E_SEQ_GENERAL.BUSY:;
	CASE THIS^.stSeqCtrlGeneral.iInternalSeqStateCase OF
    0:  // Nest 1 stop and low pressure pump bypass
      IF TRUE 
			AND THIS^.itfNest1.M_Stop()
      AND THIS^.itfLowPressurePump.M_Bypass(bEnable:= TRUE)
			THEN 
        PrgMeasure.bRecord := FALSE;
				THIS^.stSeqCtrlGeneral.iInternalSeqStateCase := 10; 
			END_IF
      
    10:  // Nest 2-4 stop
      IF TRUE 
			AND THIS^.itfNest2.M_Stop()
			AND THIS^.itfNest3.M_Stop()
			AND THIS^.itfNest4.M_Stop()
			THEN 
				THIS^.stSeqCtrlGeneral.iInternalSeqStateCase := 1000; 
			END_IF
      
    1000: // Exit step
      IF TRUE
      AND THIS^.itfTimerNest1.M_StopTimer()
      AND THIS^.itfTimerNest2.M_StopTimer()
      AND THIS^.itfTimerNest3.M_StopTimer()
      AND THIS^.itfTimerNest4.M_StopTimer()
			THEN 
				THIS^.stSeqCtrlGeneral.iInternalSeqStateCase := 9999; 
			END_IF
      
	ELSE
		THIS^.stSeqCtrlGeneral.eActiveSeqState := E_SEQ_GENERAL.DONE;  
	END_CASE
	THIS^.stSeqCtrlGeneral.strExtraInfo := CONCAT('Internal state: ', TO_STRING(THIS^.stSeqCtrlGeneral.iInternalSeqStateCase));
E_SEQ_GENERAL.DONE:;
E_SEQ_GENERAL.ERROR:;
E_SEQ_GENERAL.TIME_OUT:; 

IF TRUE
AND THIS^.stSeqCtrlGeneral.bTimeOutActiveQuit 
THEN
  THIS^.stSeqCtrlGeneral.strExtraInfo := 'Bitte quittieren und erneut testen';
  IF TRUE
  //AND itfOpMode.P_QUIT
  THEN
    THIS^.stSeqCtrlGeneral.eActiveSeqState := E_SEQ_GENERAL.EXECUTE;
	END_IF
  
END_IF

ELSE
  THIS^.stSeqCtrlGeneral.eActiveSeqState := E_SEQ_GENERAL.ERROR;
END_CASE
END_METHOD

METHOD PRIVATE _m_Seq_STOP_ENGINE : E_SEQ_PROCESS
VAR_INPUT
END_VAR
VAR
	ActiveSeq: STRING;
END_VAR
VAR
	
END_VAR
//THIS^._m_GeneralStepSetting(StepType:=E_STEP_STATE_TYPE.INIT,
ActiveSeq := TO_STRING(THIS^.eSeq);

CASE THIS^.stSeqCtrlGeneral.eActiveSeqState OF
E_SEQ_GENERAL.READY:;

	
E_SEQ_GENERAL.EXECUTE:;
	IF TRUE
	AND _m_Delay(T#1S)
	THEN
		THIS^.stSeqCtrlGeneral.eActiveSeqState := E_SEQ_GENERAL.RESET;
	END_IF
E_SEQ_GENERAL.RESET:;
	stSeqCtrlGeneral.iInternalSeqStateCase := 0;
  
	IF TRUE
	THEN
		THIS^.stSeqCtrlGeneral.eActiveSeqState := E_SEQ_GENERAL.BUSY;
	END_IF
E_SEQ_GENERAL.BUSY:;
	CASE THIS^.stSeqCtrlGeneral.iInternalSeqStateCase OF
		0:  // Nest 1 engine stop
      IF TRUE 
			AND THIS^.itfNest1.M_StopEngine()
			THEN 
				THIS^.stSeqCtrlGeneral.iInternalSeqStateCase := 10; 
			END_IF
      
    10: // Nest 2-4 engine stop
      IF TRUE 
			AND THIS^.itfNest2.M_StopEngine()
			AND THIS^.itfNest3.M_StopEngine()
			AND THIS^.itfNest4.M_StopEngine()
			THEN 
				THIS^.stSeqCtrlGeneral.iInternalSeqStateCase := 1000; 
			END_IF
      
    1000: // Exit step
      IF TRUE
      AND THIS^.itfTimerNest1.M_StopTimer()
      AND THIS^.itfTimerNest2.M_StopTimer()
      AND THIS^.itfTimerNest3.M_StopTimer()
      AND THIS^.itfTimerNest4.M_StopTimer()
			THEN 
				THIS^.stSeqCtrlGeneral.iInternalSeqStateCase := 9999; 
			END_IF
      
	ELSE
		THIS^.stSeqCtrlGeneral.eActiveSeqState := E_SEQ_GENERAL.DONE;  
	END_CASE
	THIS^.stSeqCtrlGeneral.strExtraInfo := CONCAT('Internal state: ', TO_STRING(THIS^.stSeqCtrlGeneral.iInternalSeqStateCase));
E_SEQ_GENERAL.DONE:;
E_SEQ_GENERAL.ERROR:;
E_SEQ_GENERAL.TIME_OUT:; 

IF TRUE
AND THIS^.stSeqCtrlGeneral.bTimeOutActiveQuit 
THEN
  THIS^.stSeqCtrlGeneral.strExtraInfo := 'Bitte quittieren und erneut testen';
  IF TRUE
  //AND itfOpMode.P_QUIT
  THEN
    THIS^.stSeqCtrlGeneral.eActiveSeqState := E_SEQ_GENERAL.EXECUTE;
	END_IF
  
END_IF

ELSE
  THIS^.stSeqCtrlGeneral.eActiveSeqState := E_SEQ_GENERAL.ERROR;
END_CASE
END_METHOD

METHOD PRIVATE _m_SequenceManager
VAR_INPUT
END_VAR
IF FALSE
//AND THIS^.eActiveSeqState=DONE 
AND eLastSeq<>eSeq
THEN
	IF THIS^.stSeqCtrlGeneral.eActiveSeqState<>E_SEQ_GENERAL.EXECUTE THEN
		THIS^.stSeqCtrlGeneral.eActiveSeqState:=E_SEQ_GENERAL.READY;
	END_IF
END_IF

eSeq := eNextSeq;

//DelayTimer und TimeOut Timer verwalten
stSeqCtrlGeneral.bActiveStep:=	TRUE
				AND eLastSeq					=	eSeq
				AND stSeqCtrlGeneral.eLastActiveSeqState			=	stSeqCtrlGeneral.eActiveSeqState
				AND	stSeqCtrlGeneral.iLastInternalSeqStateCase	=	stSeqCtrlGeneral.iInternalSeqStateCase
				;
			
IF NOT stSeqCtrlGeneral.bActiveStep THEN
	stSeqCtrlGeneral.bDelayActive:=FALSE;
	stSeqCtrlGeneral.bTimeOutActiveQuit:=FALSE;
	stSeqCtrlGeneral.bTimeOutActiveNoQuit:=FALSE;
  THIS^.stSeqCtrlGeneral.strExtraInfo:='';
END_IF

_m_SaveLastStep();
stSeqCtrlGeneral.tonDelay	(IN:=stSeqCtrlGeneral.bActiveStep AND stSeqCtrlGeneral.bDelayActive, 		PT:=stSeqCtrlGeneral.tDelay);
stSeqCtrlGeneral.tonTimeOut	(IN:=stSeqCtrlGeneral.bActiveStep AND (stSeqCtrlGeneral.bTimeOutActiveNoQuit OR stSeqCtrlGeneral.bTimeOutActiveQuit), 	PT:=stSeqCtrlGeneral.tTimeOut);
stSeqCtrlGeneral.tonStepTime	(IN:= stSeqCtrlGeneral.bActiveStep, PT:= T#24H);

IF stSeqCtrlGeneral.tonTimeOut.Q  THEN
	stSeqCtrlGeneral.eActiveSeqState:=E_SEQ_GENERAL.TIME_OUT;
END_IF

IF stSeqCtrlGeneral.iError<>0 THEN
	eSeq:=E_SEQ_PROCESS.ERROR_SEQ;
END_IF



eLastSeq					:=	eSeq;
stSeqCtrlGeneral.eLastActiveSeqState			:=	stSeqCtrlGeneral.eActiveSeqState;
stSeqCtrlGeneral.iLastInternalSeqStateCase	:=	stSeqCtrlGeneral.iInternalSeqStateCase;

// Reset set ready state
IF THIS^.stSeqCtrlGeneral.bExitSetReadyState THEN
  THIS^.stSeqCtrlGeneral.bExitSetReadyState := FALSE;
END_IF
END_METHOD

METHOD PRIVATE _m_TimeOut : BOOL
VAR_INPUT
	bTimeoutActiveToQuit:	BOOL;
	bTimeOutActiveNoQuit:	BOOL;
	tTimeOut:				TIME;	
END_VAR
THIS^.stSeqCtrlGeneral.bTimeOutActiveQuit:=	bTimeoutActiveToQuit;
THIS^.stSeqCtrlGeneral.bTimeOutActiveNoQuit:=	bTimeOutActiveNoQuit;
THIS^.stSeqCtrlGeneral.tTimeOut:=			tTimeOut;
_m_TimeOut:=FALSE;
IF THIS^.stSeqCtrlGeneral.tonTimeOut.Q THEN
	_m_TimeOut:=TRUE;
END_IF
END_METHOD

METHOD FB_init : BOOL
VAR_INPUT
	bInitRetains : BOOL; // if TRUE, the retain variables are initialized (warm start / cold start)
	bInCopyCode : BOOL;  // if TRUE, the instance afterwards gets moved into the copy code (online change)
  
  itfOpMode:											                        I_OP_MODE; 
  itfEventLogger:                                         I_EVENT_LOGGER; 
  itfTimerNest1:                                          I_CLOCK; 
  itfTimerNest2:                                          I_CLOCK; 
  itfTimerNest3:                                          I_CLOCK; 
  itfTimerNest4:                                          I_CLOCK;
  itfNest1:                                               I_PROCESS_NEST1;
  itfNest2:                                               I_PROCESS_NEST2_4;
  itfNest3:                                               I_PROCESS_NEST2_4;
  itfNest4:                                               I_PROCESS_NEST2_4;
  itfLowPressurePump:                                     I_PUMP_WITH_BYPASS;
  itfOilCooler:                                           I_PUMP;
  itfBypassPump:                                          I_PUMP;
  itfLevelSwitch_AggregateTank1_Out1:                     I_BINARY_SWITCH;
  itfLevelSwitch_AggregateTank1_Out2:                     I_BINARY_SWITCH;
  itfTemperatureSwitch_AggregateTank1_Out1:               I_BINARY_SWITCH;
  itfTemperatureSwitch_AggregateTank1_Out2:               I_BINARY_SWITCH;
  itfLevelSwitch_AggregateTank2_Out1:                     I_BINARY_SWITCH;
  itfLevelSwitch_AggregateTank2_Out2:                     I_BINARY_SWITCH;
  itfLevelSwitch_AggregateTank2_Out3:                     I_BINARY_SWITCH;
  itfSwitch_AggregateFilter_Dirty:                        I_BINARY_SWITCH; 
END_VAR
THIS^.itfOpMode := itfOpMode;
THIS^.itfEventLogger := itfEventLogger;
THIS^.itfTimerNest1 := itfTimerNest1;
THIS^.itfTimerNest2 := itfTimerNest2;
THIS^.itfTimerNest3 := itfTimerNest3;
THIS^.itfTimerNest4 := itfTimerNest4;
THIS^.itfNest1 := itfNest1;
THIS^.itfNest2 := itfNest2;
THIS^.itfNest3 := itfNest3;
THIS^.itfNest4 := itfNest4;
THIS^.itfLowPressurePump := itfLowPressurePump;
THIS^.itfOilCooler := itfOilCooler;
THIS^.itfBypassPump := itfBypassPump;
THIS^.itfLevelSwitch_AggregateTank1_Out1 := itfLevelSwitch_AggregateTank1_Out1;
THIS^.itfLevelSwitch_AggregateTank1_Out2 := itfLevelSwitch_AggregateTank1_Out2;
THIS^.itfTemperatureSwitch_AggregateTank1_Out1 := itfTemperatureSwitch_AggregateTank1_Out1;
THIS^.itfTemperatureSwitch_AggregateTank1_Out2 := itfTemperatureSwitch_AggregateTank1_Out2;
THIS^.itfLevelSwitch_AggregateTank2_Out1 := itfLevelSwitch_AggregateTank2_Out1;
THIS^.itfLevelSwitch_AggregateTank2_Out2 := itfLevelSwitch_AggregateTank2_Out2;
THIS^.itfLevelSwitch_AggregateTank2_Out3 := itfLevelSwitch_AggregateTank2_Out3;
THIS^.itfSwitch_AggregateFilter_Dirty := itfSwitch_AggregateFilter_Dirty;
END_METHOD

METHOD M_BreakPressureDet : BOOL
VAR_INPUT
  stBreakPressureParams:                 ST_RECIPE_BREAK_PRESSURE;
END_VAR
M_BreakPressureDet := THIS^.stSeqCtrlGeneral.eActiveSeqState = E_SEQ_GENERAL.DONE;

// Assign input
THIS^.stBPDParams := stBreakPressureParams;

// General
IF THIS^.stSeqCtrlGeneral.eActiveSeqState = E_SEQ_GENERAL.READY THEN
  THIS^.eNextSeq := E_SEQ_PROCESS.BREAK_PRESSURE_DET;
  THIS^.stSeqCtrlGeneral.eActiveSeqState := E_SEQ_GENERAL.EXECUTE;
END_IF
END_METHOD

METHOD M_EnduranceRun : BOOL
VAR_INPUT
  stEnduranceRunParams:                 ST_RECIPE_ENDURANCE_RUN;
END_VAR
M_EnduranceRun := THIS^.stSeqCtrlGeneral.eActiveSeqState = E_SEQ_GENERAL.DONE;

// Assign input
THIS^.stERParams := stEnduranceRunParams;

// General
IF THIS^.stSeqCtrlGeneral.eActiveSeqState = E_SEQ_GENERAL.READY THEN
  THIS^.eNextSeq := E_SEQ_PROCESS.ENDURANCE_RUN;
  THIS^.stSeqCtrlGeneral.eActiveSeqState := E_SEQ_GENERAL.EXECUTE;
END_IF
END_METHOD

METHOD M_EStop : BOOL
M_EStop := THIS^.stSeqCtrlGeneral.eActiveSeqState = E_SEQ_GENERAL.DONE;

IF THIS^.stSeqCtrlGeneral.eActiveSeqState = E_SEQ_GENERAL.READY THEN
  THIS^.eNextSeq := E_SEQ_PROCESS.ESTOP;
  THIS^.stSeqCtrlGeneral.eActiveSeqState := E_SEQ_GENERAL.EXECUTE;
END_IF
END_METHOD

METHOD M_LeakTest1 : BOOL
VAR_INPUT
  stLeakTest1Params:                 ST_RECIPE_LEAK_TEST1;
END_VAR
M_LeakTest1 := THIS^.stSeqCtrlGeneral.eActiveSeqState = E_SEQ_GENERAL.DONE;

// Assign input
THIS^.stLT1Params := stLeakTest1Params;

// General
IF THIS^.stSeqCtrlGeneral.eActiveSeqState = E_SEQ_GENERAL.READY THEN
  THIS^.eNextSeq := E_SEQ_PROCESS.LEAK_TEST_1;
  THIS^.stSeqCtrlGeneral.eActiveSeqState := E_SEQ_GENERAL.EXECUTE;
END_IF
END_METHOD

METHOD M_LeakTest2 : BOOL
VAR_INPUT
  stLeakTest2Params:                 ST_RECIPE_LEAK_TEST2;
END_VAR
M_LeakTest2 := THIS^.stSeqCtrlGeneral.eActiveSeqState = E_SEQ_GENERAL.DONE;

// Assign input
THIS^.stLT2Params := stLeakTest2Params;

// General
IF THIS^.stSeqCtrlGeneral.eActiveSeqState = E_SEQ_GENERAL.READY THEN
  THIS^.eNextSeq := E_SEQ_PROCESS.LEAK_TEST_2;
  THIS^.stSeqCtrlGeneral.eActiveSeqState := E_SEQ_GENERAL.EXECUTE;
END_IF
END_METHOD

METHOD M_Reset : BOOL
M_Reset := THIS^.stSeqCtrlGeneral.eActiveSeqState = E_SEQ_GENERAL.DONE;

IF THIS^.stSeqCtrlGeneral.eActiveSeqState = E_SEQ_GENERAL.READY THEN
  THIS^.eNextSeq := E_SEQ_PROCESS.INIT;
  THIS^.stSeqCtrlGeneral.eActiveSeqState := E_SEQ_GENERAL.EXECUTE;
END_IF
END_METHOD

{warning 'Methodenimplementierung hinzufügen'}
(*=== Method: M_Run  ============================================

 @brief: Here is the global code (Timer, Event, Flange,...)*)
METHOD M_Run
END_METHOD

METHOD M_SetReady : BOOL
VAR_INPUT
  
END_VAR
M_SetReady := TRUE
              AND THIS^.stSeqCtrlGeneral.eActiveSeqState = E_SEQ_GENERAL.READY
              AND THIS^.eSeq = E_SEQ_PROCESS.BASE;

THIS^.stSeqCtrlGeneral.eActiveSeqState := E_SEQ_GENERAL.READY;
THIS^.eNextSeq := E_SEQ_PROCESS.BASE;
END_METHOD

METHOD M_Stop : BOOL
M_Stop := THIS^.stSeqCtrlGeneral.eActiveSeqState = E_SEQ_GENERAL.DONE;

IF THIS^.stSeqCtrlGeneral.eActiveSeqState = E_SEQ_GENERAL.READY THEN
  THIS^.eNextSeq := E_SEQ_PROCESS.STOP;
  THIS^.stSeqCtrlGeneral.eActiveSeqState := E_SEQ_GENERAL.EXECUTE;
END_IF
END_METHOD

METHOD M_StopEngine : BOOL
M_StopEngine := THIS^.stSeqCtrlGeneral.eActiveSeqState = E_SEQ_GENERAL.DONE;

IF THIS^.stSeqCtrlGeneral.eActiveSeqState = E_SEQ_GENERAL.READY THEN
  THIS^.eNextSeq := E_SEQ_PROCESS.STOP_ENGINE;
  THIS^.stSeqCtrlGeneral.eActiveSeqState := E_SEQ_GENERAL.EXECUTE;
END_IF
END_METHOD

{warning 'Eigenschaftenimplementierung hinzufügen'}
PROPERTY P_CurrentCycleNest1 : UDINT
GET
P_CurrentCycleNest1 := THIS^.udiCurrentCyclesNest1;
END_GET
END_PROPERTY

{warning 'Eigenschaftenimplementierung hinzufügen'}
PROPERTY P_CurrentCycleNest2 : UDINT
GET
P_CurrentCycleNest2 := THIS^.udiCurrentCyclesNest2;
END_GET
END_PROPERTY

{warning 'Eigenschaftenimplementierung hinzufügen'}
PROPERTY P_CurrentCycleNest3 : UDINT
GET
P_CurrentCycleNest3 := THIS^.udiCurrentCyclesNest3;
END_GET
END_PROPERTY

{warning 'Eigenschaftenimplementierung hinzufügen'}
PROPERTY P_CurrentCycleNest4 : UDINT
GET
P_CurrentCycleNest4 := THIS^.udiCurrentCyclesNest4;
END_GET
END_PROPERTY

{warning 'Eigenschaftenimplementierung hinzufügen'}
(*=== Property: P_Event  ============================================

 @param [set]: 	Set the Structure "ST_EVENT" from another Object
 @param [get]: 	Return the Structure "ST_EVENT", it contains the actual 
					event of the Object *)
PROPERTY P_Event : GenLib.ST_EVENT
GET
END_GET
SET
END_SET
END_PROPERTY

{warning 'Eigenschaftenimplementierung hinzufügen'}
(*=== Property: P_FullObjectPath  ============================================

 @param [set]: 	Set the Object Path (Clear String of Object)
 @param [get]: 	Return the Objectpath *)
PROPERTY P_FullObjectPath : STRING
GET
END_GET
SET
END_SET
END_PROPERTY

{warning 'Eigenschaftenimplementierung hinzufügen'}
(*=== Property: P_Global_Ack  ============================================

 @param [set]: 	Set the Bit for Ack from another Object
 @param [get]: 	Return the state of Ack Bit*)
PROPERTY P_Global_Ack : BOOL
GET
END_GET
SET
END_SET
END_PROPERTY

{warning 'Eigenschaftenimplementierung hinzufügen'}
(*=== Property: P_GlobalID  ============================================

 @param [set]: 	-
 @param [get]: 	Return the string of instance path*)
PROPERTY P_GlobalID : STRING
GET
END_GET
END_PROPERTY

{warning 'Eigenschaftenimplementierung hinzufügen'}
PROPERTY P_ReadyState : BOOL
GET
P_ReadyState := THIS^.stSeqCtrlGeneral.eActiveSeqState = E_SEQ_GENERAL.READY;
END_GET
END_PROPERTY

END_FUNCTION_BLOCK

// ---- FUNCTIONS/FUNCTIONS/MATH/F_RoundLREAL.TcPOU
FUNCTION F_RoundLREAL : LREAL
VAR_INPUT
	lrValue:					LREAL;
	uiDezimalPlace:	UINT;
END_VAR
VAR
	lrResult:				REAL;
	uiMultiplier:		UINT := 1;
	i:							UINT;
END_VAR

FOR i := 1 TO uiDezimalPlace BY 1 DO
	uiMultiplier := uiMultiplier * 10;
END_FOR

lrResult := TO_REAL(TO_DINT(lrValue * uiMultiplier)) / uiMultiplier;

F_RoundLREAL := lrResult;

END_FUNCTION

// ---- MODULE/ACTOR_VALVE/PNEUMATIC_ACTOR/POU/FB_STOP_GATE.TcPOU
{attribute 'reflection'} 
{attribute 'no_explicit_call' := 'do not call this POU directly'} 
FUNCTION_BLOCK FB_STOP_GATE IMPLEMENTS I_STOP_GATE
VAR_INPUT
END_VAR
VAR_OUTPUT
END_VAR
VAR
	{attribute 'instance-path'} 
    {attribute 'noinit'} 
	strInstancePath: STRING;
	strFullObjectPath: STRING;
	stEvent: ST_EVENT;
	bAck: BOOL;
	itfOpMode:				I_OP_MODE;
	itfValveOpenStopGate:	I_BASE_VALVE;
	itfSensorByStopGate: 	I_BINARY_SWITCH;
	itfSensorCongestion: 	I_BINARY_SWITCH;
	
	tonToBase: Tc2_Standard.TON;
	tToBase: TIME;
	tonToWork: Tc2_Standard.TON;
	tToWork: TIME;
	bViewToBase: BOOL;
	bViewToWork: BOOL;
	
	
END_VAR

METHOD FB_init : BOOL
VAR_INPUT
	bInitRetains : BOOL; // if TRUE, the retain variables are initialized (warm start / cold start)
	bInCopyCode : BOOL;  // if TRUE, the instance afterwards gets moved into the copy code (online change)
END_VAR
END_METHOD

{warning 'Methodenimplementierung hinzufügen'}
METHOD M_Close
END_METHOD

{warning 'Methodenimplementierung hinzufügen'}
METHOD M_Open
END_METHOD

{warning 'Methodenimplementierung hinzufügen'}
(*=== Method: M_Run  ============================================

 @brief: Here is the global code (Timer, Event, Flange,...)*)
METHOD M_Run
END_METHOD

{warning 'Methodenimplementierung hinzufügen'}
METHOD M_Seperate
VAR_INPUT
	iCntCarrier	: INT;
END_VAR
END_METHOD


PROPERTY P_CarrierByStopGate : BOOL
GET
END_GET
END_PROPERTY


PROPERTY P_Congestion : BOOL
GET
END_GET
END_PROPERTY


(*=== Property: P_Event  ============================================

 @param [set]: 	Set the Structure "ST_EVENT" from another Object
 @param [get]: 	Return the Structure "ST_EVENT", it contains the actual 
					event of the Object *)
PROPERTY P_Event : ST_EVENT
GET
END_GET
SET
END_SET
END_PROPERTY


(*=== Property: P_FullObjectPath  ============================================

 @param [set]: 	Set the Object Path (Clear String of Object)
 @param [get]: 	Return the Objectpath *)
PROPERTY P_FullObjectPath : STRING
GET
END_GET
SET
END_SET
END_PROPERTY


(*=== Property: P_Global_Ack  ============================================

 @param [set]: 	Set the Bit for Ack from another Object
 @param [get]: 	Return the state of Ack Bit*)
PROPERTY P_Global_Ack : BOOL
GET
END_GET
SET
END_SET
END_PROPERTY


(*=== Property: P_GlobalID  ============================================

 @param [set]: 	-
 @param [get]: 	Return the string of instance path*)
PROPERTY P_GlobalID : STRING
GET
END_GET
END_PROPERTY

END_FUNCTION_BLOCK

// ---- MODULE/ACTOR_VALVE/PNEUMATIC_ACTOR/POU/FB_VAC_BLOW_VALVE.TcPOU
{attribute 'reflection'} 
{attribute 'no_explicit_call' := 'do not call this POU directly'} 
FUNCTION_BLOCK FB_VAC_BLOW_VALVE IMPLEMENTS I_VAC_VALVE
VAR_INPUT
END_VAR
VAR_OUTPUT
END_VAR
VAR
	{attribute 'instance-path'} 
    {attribute 'noinit'} 
	strInstancePath: STRING;
	strFullObjectPath: STRING;
	stEvent: ST_EVENT;
	bAck: BOOL;
	itfOpMode:			I_OP_MODE;
	itfValveVac: I_BASE_VALVE;
	itfValveBlow: I_BASE_VALVE;
	itfSensorVacDetect: I_BINARY_SWITCH;

	
END_VAR

METHOD FB_init : BOOL
VAR_INPUT
	bInitRetains : BOOL; // if TRUE, the retain variables are initialized (warm start / cold start)
	bInCopyCode : BOOL;  // if TRUE, the instance afterwards gets moved into the copy code (online change)
	itfOpMode:			I_OP_MODE;
	itfValveVac: I_BASE_VALVE;
	itfValveBlow: I_BASE_VALVE;
	itfSensorVacDetect: I_BINARY_SWITCH;
END_VAR
THIS^.itfOpMode:= itfOpMode;
THIS^.itfValveVac:= itfValveVac;
THIS^.itfValveBlow:= itfValveBlow;
THIS^.itfSensorVacDetect:= itfSensorVacDetect;
END_METHOD

{warning 'Methodenimplementierung hinzufügen'}
METHOD M_AllOff
THIS^.itfValveVac.M_Close();
THIS^.itfValveBlow.M_Close();
END_METHOD

{warning 'Methodenimplementierung hinzufügen'}
METHOD M_Blow
THIS^.itfValveVac.M_Close();
THIS^.itfValveBlow.M_OPEN();
END_METHOD

{warning 'Methodenimplementierung hinzufügen'}
(*=== Method: M_Run  ============================================

 @brief: Here is the global code (Timer, Event, Flange,...)*)
METHOD M_Run
F_HandleInheritanceObjectInMRun(itfInheritanceObject:=THIS^.itfSensorVacDetect,itfThisObject:=THIS^);
F_HandleInheritanceObjectInMRun(itfInheritanceObject:=THIS^.itfValveVac,itfThisObject:=THIS^);
END_METHOD

{warning 'Methodenimplementierung hinzufügen'}
METHOD M_Vac
THIS^.itfValveVac.M_OPEN();
THIS^.itfValveBlow.M_Close();
END_METHOD


(*=== Property: P_Event  ============================================

 @param [set]: 	Set the Structure "ST_EVENT" from another Object
 @param [get]: 	Return the Structure "ST_EVENT", it contains the actual 
					event of the Object *)
PROPERTY P_Event : ST_EVENT
GET
P_Event:= stEvent;
END_GET
SET
END_SET
END_PROPERTY


(*=== Property: P_FullObjectPath  ============================================

 @param [set]: 	Set the Object Path (Clear String of Object)
 @param [get]: 	Return the Objectpath *)
PROPERTY P_FullObjectPath : STRING
GET
P_FullObjectPath:= THIS^.strFullObjectPath;
END_GET
SET
THIS^.strFullObjectPath:= P_FullObjectPath;
END_SET
END_PROPERTY


(*=== Property: P_Global_Ack  ============================================

 @param [set]: 	Set the Bit for Ack from another Object
 @param [get]: 	Return the state of Ack Bit*)
PROPERTY P_Global_Ack : BOOL
GET
P_Global_Ack:= THIS^.bAck;
END_GET
SET
THIS^.bAck:=P_Global_Ack;
END_SET
END_PROPERTY


(*=== Property: P_GlobalID  ============================================

 @param [set]: 	-
 @param [get]: 	Return the string of instance path*)
PROPERTY P_GlobalID : STRING
GET
P_GlobalID:= THIS^.strInstancePath;
END_GET
END_PROPERTY


PROPERTY P_STATE : E_PNEU_VAC_VALVE
GET
IF THIS^.itfValveVac.P_IS_OPEN THEN
	P_STATE:=E_PNEU_VAC_VALVE.Vac_ON_NotDetect;
END_IF

IF THIS^.itfValveVac.P_IS_CLOSE THEN
	P_STATE:=E_PNEU_VAC_VALVE.AllOff;
END_IF

IF THIS^.itfSensorVacDetect.P_Active THEN
	 P_STATE:=E_PNEU_VAC_VALVE.VacDetect;
 END_IF
 
 IF THIS^.itfValveBlow.P_IS_OPEN THEN
	 P_STATE:=E_PNEU_VAC_VALVE.Blowing;
 END_IF
END_GET
END_PROPERTY

END_FUNCTION_BLOCK

// ---- MODULE/ACTOR_VALVE/PNEUMATIC_ACTOR/POU/FB_VAC_VALVE.TcPOU
{attribute 'reflection'} 
{attribute 'no_explicit_call' := 'do not call this POU directly'} 
FUNCTION_BLOCK FB_VAC_VALVE IMPLEMENTS I_VAC_VALVE
VAR_INPUT
END_VAR
VAR_OUTPUT
END_VAR
VAR
	{attribute 'instance-path'} 
    {attribute 'noinit'} 
	strInstancePath: STRING;
	strFullObjectPath: STRING;
	stEvent: ST_EVENT;
	bAck: BOOL;
	itfOpMode:			I_OP_MODE;
	itfValveVac: I_BASE_VALVE;
	itfSensorVacDetect: I_BINARY_SWITCH;

	
END_VAR

METHOD FB_init : BOOL
VAR_INPUT
	bInitRetains : BOOL; // if TRUE, the retain variables are initialized (warm start / cold start)
	bInCopyCode : BOOL;  // if TRUE, the instance afterwards gets moved into the copy code (online change)
	itfOpMode:	I_OP_MODE;
	itfValveVac: I_BASE_VALVE;
	itfSensorVacDetect: I_BINARY_SWITCH;
END_VAR
THIS^.itfOpMode:= itfOpMode;
THIS^.itfValveVac:= itfValveVac;
THIS^.itfSensorVacDetect:= itfSensorVacDetect;
END_METHOD

{warning 'Methodenimplementierung hinzufügen'}
METHOD M_AllOff
THIS^.itfValveVac.M_Close();
END_METHOD

{warning 'Methodenimplementierung hinzufügen'}
METHOD M_Blow
THIS^.itfValveVac.M_Close();
END_METHOD

{warning 'Methodenimplementierung hinzufügen'}
(*=== Method: M_Run  ============================================

 @brief: Here is the global code (Timer, Event, Flange,...)*)
METHOD M_Run
F_HandleInheritanceObjectInMRun(itfInheritanceObject:=THIS^.itfSensorVacDetect,itfThisObject:=THIS^);
F_HandleInheritanceObjectInMRun(itfInheritanceObject:=THIS^.itfValveVac,itfThisObject:=THIS^);
END_METHOD

{warning 'Methodenimplementierung hinzufügen'}
METHOD M_Vac
THIS^.itfValveVac.M_OPEN();
END_METHOD


(*=== Property: P_Event  ============================================

 @param [set]: 	Set the Structure "ST_EVENT" from another Object
 @param [get]: 	Return the Structure "ST_EVENT", it contains the actual 
					event of the Object *)
PROPERTY P_Event : ST_EVENT
GET
P_Event:= stEvent;
END_GET
SET
END_SET
END_PROPERTY


(*=== Property: P_FullObjectPath  ============================================

 @param [set]: 	Set the Object Path (Clear String of Object)
 @param [get]: 	Return the Objectpath *)
PROPERTY P_FullObjectPath : STRING
GET
P_FullObjectPath:= THIS^.strFullObjectPath;
END_GET
SET
THIS^.strFullObjectPath:= P_FullObjectPath;
END_SET
END_PROPERTY


(*=== Property: P_Global_Ack  ============================================

 @param [set]: 	Set the Bit for Ack from another Object
 @param [get]: 	Return the state of Ack Bit*)
PROPERTY P_Global_Ack : BOOL
GET
P_Global_Ack:= THIS^.bAck;
END_GET
SET
THIS^.bAck:=P_Global_Ack;
END_SET
END_PROPERTY


(*=== Property: P_GlobalID  ============================================

 @param [set]: 	-
 @param [get]: 	Return the string of instance path*)
PROPERTY P_GlobalID : STRING
GET
P_GlobalID:= THIS^.strInstancePath;
END_GET
END_PROPERTY


PROPERTY P_STATE : E_PNEU_VAC_VALVE
GET
IF THIS^.itfValveVac.P_IS_OPEN THEN
	P_STATE:=E_PNEU_VAC_VALVE.Vac_ON_NotDetect;
END_IF

IF THIS^.itfValveVac.P_IS_CLOSE THEN
	P_STATE:=E_PNEU_VAC_VALVE.AllOff;
END_IF

IF THIS^.itfSensorVacDetect.P_Active THEN
	 P_STATE:=E_PNEU_VAC_VALVE.VacDetect;
 END_IF
END_GET
END_PROPERTY

END_FUNCTION_BLOCK

// ---- MODULE/ACTOR_VALVE/PNEUMATIC_ACTOR/POU/FB_VISU_CYLINDER.TcPOU
FUNCTION_BLOCK FB_VISU_CYLINDER
VAR_INPUT
END_VAR
VAR_OUTPUT
END_VAR
VAR
	itfPneuActor: I_PNEU_ACTOR;	
	itfOpMode: I_OP_MODE;
	iMove: INT;
	iNegMove: INT;
	iMoveSmall: INT;
	iNegMoveSmall: INT;
	iAngle: INT;
	iNegAngle: INT;
	strInfo: STRING;
	strFullObjName: STRING;
	bMoveToBase: BOOL;
	bMoveToWork: BOOL;
	bAllOff: BOOL;
	bInBasePos: BOOL;
	bInWorkPos: BOOL;
	bInMidPos: 	BOOL;
	bFaultWorkPos: BOOL;
	bFaultBasePos: BOOL;
	dwFrameColorBase: DWORD:= 16#FF00BFFF;
	dwFrameColorWork: DWORD:= 16#FF00BFFF;
	dwFrameColorMid: DWORD:= 16#FF00BFFF;
	bBaseArrowInvisible: BOOL:=TRUE;
	bWorkArrowInvisible: BOOL:=TRUE;
	bMidkArrowInvisible: BOOL:=TRUE;
	iFrame: INT;
	bFrameInvisible: BOOL:= TRUE;
	stEvent: ST_EVENT;
	dwColor: DWORD;
END_VAR

IF NOT (itfOpMode.P_OP_MODE_STATE=OP_MODE.MANUAL) THEN
	bFrameInvisible:= TRUE;
END_IF

IF (itfPneuActor.P_State=E_POS_STATE.MoveToBase) THEN
//IF bMoveToBase AND NOT bInBasePos THEN
	iMove:=-30;
	iAngle:=-90;
	//strInfo:= 'Zylinder fährt in Grundposition';
	strInfo:= F_RET_TXTLIST_ENTRY(strPortNr:= '851', strID:='3', strTxtLstName:= 'TXT_LIST_PNEMATIC_ACTOR');
	//bMoveToWork:= FALSE;
	dwFrameColorBase:= 16#FFFFA500;
	bBaseArrowInvisible:= FALSE;
	bWorkArrowInvisible:=TRUE;	
	bMidkArrowInvisible:=TRUE;
END_IF

IF (itfPneuActor.P_State=E_POS_STATE.InBasePos) THEN
//IF bMoveToBase AND bInBasePos THEN
	iMove:=0;
	iAngle:=0;
	//strInfo:= 'Zylinder ist in Grundposition';
	strInfo:= F_RET_TXTLIST_ENTRY(strPortNr:= '851', strID:='4', strTxtLstName:= 'TXT_LIST_PNEMATIC_ACTOR');
	//bMoveToWork:= FALSE;
	dwFrameColorBase:= 16#FF77BB77;
	bBaseArrowInvisible:= FALSE;
	bWorkArrowInvisible:=TRUE;	
	bMidkArrowInvisible:=TRUE;
END_IF

IF (itfPneuActor.P_State=E_POS_STATE.MoveToWork) THEN
//IF bMoveToWork AND NOT bInworkPos THEN
	iMove:=-30;
	iAngle:=-90;
	//strInfo:= 'Zylinder fährt in Arbeitsposition';
	strInfo:= F_RET_TXTLIST_ENTRY(strPortNr:= '851', strID:='5', strTxtLstName:= 'TXT_LIST_PNEMATIC_ACTOR');
	//bMoveToBase:= FALSE;
	dwFrameColorwork:= 16#FFFFA500;
	bBaseArrowInvisible:= TRUE;
	bWorkArrowInvisible:=FALSE;	
	bMidkArrowInvisible:=TRUE;
END_IF

IF (itfPneuActor.P_State=E_POS_STATE.InWorkPos) THEN
//IF bMoveToWork AND bInWorkPos THEN
	iMove:=-70;
	iAngle:=180;
	//strInfo:= 'Zylinder ist in Arbeitsposition';
	strInfo:= F_RET_TXTLIST_ENTRY(strPortNr:= '851', strID:='6', strTxtLstName:= 'TXT_LIST_PNEMATIC_ACTOR');
	//bMoveTobase:= FALSE;
	dwFrameColorWork:= 16#FF77BB77;
	bBaseArrowInvisible:= TRUE;
	bWorkArrowInvisible:=FALSE;	
	bMidkArrowInvisible:=TRUE;
END_IF

IF (itfPneuActor.P_State=E_POS_STATE.InMidPos) THEN
//IF bMoveToWork AND bInWorkPos THEN
	iMove:=-50;
	iAngle:=-90;
	//strInfo:= 'Zylinder ist in Arbeitsposition';
	strInfo:= F_RET_TXTLIST_ENTRY(strPortNr:= '851', strID:='15', strTxtLstName:= 'TXT_LIST_PNEMATIC_ACTOR');
	//bMoveTobase:= FALSE;
	dwFrameColorMid:= 16#FF77BB77;
	bBaseArrowInvisible:= TRUE;
	bWorkArrowInvisible:=TRUE;	
	bMidkArrowInvisible:=FALSE;
END_IF

IF (itfPneuActor.P_State=E_POS_STATE.NoDefPos) THEN
//IF bMoveToWork AND bInWorkPos THEN
	iMove:=-30;
	iNegAngle:=-90;
	//strInfo:= 'Zylinder in undefinierter Position';
	strInfo:= F_RET_TXTLIST_ENTRY(strPortNr:= '851', strID:='7', strTxtLstName:= 'TXT_LIST_PNEMATIC_ACTOR');
	//bMoveTobase:= FALSE;
	dwFrameColorWork:= 16#FF77BB77;
	bBaseArrowInvisible:= TRUE;
	bWorkArrowInvisible:=TRUE;	
	bMidkArrowInvisible:=TRUE;
END_IF

IF (itfPneuActor.P_State=E_POS_STATE.TimeOutToBase) THEN
//IF bMoveToWork AND bInWorkPos THEN
	iMove:=-30;
	iAngle:=-90;
	//strInfo:= 'Timeout bei Fahrt nach Grundstellung';
	strInfo:= F_RET_TXTLIST_ENTRY(strPortNr:= '851', strID:='8', strTxtLstName:= 'TXT_LIST_PNEUMATIC_ACTOR');
	//bMoveTobase:= FALSE;
	dwFrameColorWork:= 16#FFFF00FF;
	bBaseArrowInvisible:= TRUE;
	bWorkArrowInvisible:=FALSE;	
	bMidkArrowInvisible:=TRUE;
END_IF

IF (itfPneuActor.P_State=E_POS_STATE.TimeOutToWork) THEN
//IF bMoveToWork AND bInWorkPos THEN
	iMove:=-30;	
	iAngle:=-90;
	//strInfo:= 'Timeout bei Fahrt nach Arbeitsstellung';
	strInfo:= F_RET_TXTLIST_ENTRY(strPortNr:= '851', strID:='9', strTxtLstName:= 'TXT_LIST_PNEUMATIC_ACTOR');
	//bMoveTobase:= FALSE;
	dwFrameColorWork:= 16#FFFF00FF;
	bBaseArrowInvisible:= FALSE;
	bWorkArrowInvisible:=TRUE;	
	bMidkArrowInvisible:=TRUE;
END_IF

IF  (itfPneuActor.P_State=E_POS_STATE.MoveToWorkLock) THEN
	strInfo:= stEvent.strEventText;
	dwFrameColorWork:= Color.dwRed;
	bBaseArrowInvisible:= TRUE;
	bWorkArrowInvisible:=FALSE;	
	bMidkArrowInvisible:=TRUE;
END_IF

IF (itfPneuActor.P_State=E_POS_STATE.MoveToBaseLock) THEN
	strInfo:= stEvent.strEventText;
	dwFrameColorBase:= Color.dwRed;
	bBaseArrowInvisible:= FALSE;
	bWorkArrowInvisible:=TRUE;	
	bMidkArrowInvisible:=TRUE;
END_IF

strFullObjName:= itfPneuActor.P_FullObjectPath;

IF (itfOpMode.P_OP_MODE_STATE=OP_MODE.MANUAL) THEN
	IF bMoveToBase THEN
		itfPneuActor.M_ToBasePos();
		bMoveToBase:=FALSE;
		//bMoveToWork:= FALSE;
		//bAllOff:= FALSE;
	END_IF
	IF bMoveToWork THEN
		itfPneuActor.M_ToWorkPos();
		//bMoveToBase:=FALSE;
		bMoveToWork:= FALSE;
		//bAllOff:= FALSE;
	END_IF
	IF bAllOff THEN
		itfPneuActor.M_Stop();
		//bMoveToBase:=FALSE;
		//bMoveToWork:= FALSE;
		bAllOff:= FALSE;
	END_IF
	
ELSE
	bMoveToBase:=FALSE;
	bMoveToWork:= FALSE;
    bAllOff:= FALSE;
END_IF



iNegMove:= iMove*(-1);
iNegAngle:=iAngle*(-1);
iMoveSmall:=iMove/2;
iNegMoveSmall:=iNegMove/2;
stEvent:= itfPneuActor.P_Event;

IF stEvent.bEventActive THEN
	dwColor:= Color.dwOrange;
END_IF

METHOD FB_init : BOOL
VAR_INPUT
	bInitRetains : BOOL; // if TRUE, the retain variables are initialized (warm start / cold start)
	bInCopyCode : BOOL;  // if TRUE, the instance afterwards gets moved into the copy code (online change)
	itfPneuActor: I_PNEU_ACTOR;
	itfOpMode: I_OP_MODE;
END_VAR
THIS^.itfPneuActor:= itfPneuActor;
THIS^.itfOpMode:= itfOpMode;
END_METHOD

END_FUNCTION_BLOCK

// ---- MODULE/ACTOR_VALVE/PNEUMATIC_ACTOR/POU/FB_VISU_STOP_GATE.TcPOU
FUNCTION_BLOCK FB_VISU_STOP_GATE
VAR_INPUT
END_VAR
VAR_OUTPUT
END_VAR
VAR
	iMoveCarrier: 		INT;
	bStopGateOpen: 		BOOL;
	bCarrierByStopGate: BOOL;
END_VAR

END_FUNCTION_BLOCK

// ---- MODULE/ACTOR_VALVE/PNEUMATIC_ACTOR/POU/FB_VISU_VAC_VALVE.TcPOU
FUNCTION_BLOCK FB_VISU_VAC_VALVE 
VAR_INPUT
END_VAR
VAR_OUTPUT
END_VAR
VAR
	itfVacValve: I_VAC_VALVE;
	itfOpMode: I_OP_MODE;
	strFullObjectName: STRING;
	strInfo: STRING;
	bVacOn: BOOL;
	bBlowOn: BOOL;
	bBlowOrVac: BOOL;   
	bVakOk: BOOL; 
	bActivateVac: BOOL;
	bActivateBlow: BOOL;   
	bActivateOff: BOOL;  
	bFrameInvisible: BOOL:= TRUE;
	stEvent: ST_EVENT;                                                                                                                      
END_VAR

IF NOT (itfOpMode.P_OP_MODE_STATE= OP_MODE.MANUAL) THEN
	bFrameInvisible:=TRUE;
END_IF

IF itfVacValve.P_STATE= E_PNEU_VAC_VALVE.AllOff THEN
	strInfo:= F_RET_TXTLIST_ENTRY(strPortNr:= '851', strID:='14', strTxtLstName:= 'TXT_LIST_PNEMATIC_ACTOR');
	bVacOn:=FALSE;
	bBlowOn:=FALSE;
	bVakOk:=FALSE;	
END_IF

IF itfVacValve.P_STATE= E_PNEU_VAC_VALVE.Blowing THEN
	strInfo:= F_RET_TXTLIST_ENTRY(strPortNr:= '851', strID:='13', strTxtLstName:= 'TXT_LIST_PNEMATIC_ACTOR');
	bVacOn:=FALSE;
	bBlowOn:=TRUE;	
	bVakOk:=FALSE;
END_IF

IF itfVacValve.P_STATE= E_PNEU_VAC_VALVE.Vac_ON_NotDetect THEN
	strInfo:= F_RET_TXTLIST_ENTRY(strPortNr:= '851', strID:='11', strTxtLstName:= 'TXT_LIST_PNEMATIC_ACTOR');
	bVacOn:=TRUE;
	bBlowOn:=FALSE;	
	bVakOk:=FALSE;
END_IF

IF itfVacValve.P_STATE= E_PNEU_VAC_VALVE.VacDetect THEN
	strInfo:= F_RET_TXTLIST_ENTRY(strPortNr:= '851', strID:='12', strTxtLstName:= 'TXT_LIST_PNEMATIC_ACTOR');
	bVacOn:=TRUE;
	bBlowOn:=FALSE;	
	bVakOk:=TRUE;
END_IF

strFullObjectName:= itfVacValve.P_FullObjectPath;
bBlowOrVac:=bVacOn OR bBlowOn;

IF (itfOpMode.P_OP_MODE_STATE=OP_MODE.MANUAL) THEN
	IF bActivateVac THEN
		itfVacValve.M_Vac();
	END_IF
	IF bActivateBlow THEN
		itfVacValve.M_Blow();
	END_IF
	IF bActivateOff THEN
		itfVacValve.M_AllOff();
	END_IF
ELSE
	bActivateVac:=FALSE;
	bActivateBlow:= FALSE;
	bActivateOff:= FALSE;
END_IF

stEvent:= itfVacValve.P_Event;

METHOD FB_init : BOOL
VAR_INPUT
	bInitRetains : BOOL; // if TRUE, the retain variables are initialized (warm start / cold start)
	bInCopyCode : BOOL;  // if TRUE, the instance afterwards gets moved into the copy code (online change)
	itfVacValve: I_VAC_VALVE;
	itfOpMode: I_OP_MODE;
END_VAR
THIS^.itfVacValve:= itfVacValve;
THIS^.itfOpMode:= itfOpMode;
END_METHOD

END_FUNCTION_BLOCK

// ---- MODULE/ACTOR_VALVE/PNEUMATIC_ACTOR/POU/FB_ZYLINDER_TWO_WAY.TcPOU
{attribute 'reflection'} 
{attribute 'no_explicit_call' := 'do not call this POU directly'} 
FUNCTION_BLOCK FB_ZYLINDER_TWO_WAY IMPLEMENTS I_PNEU_ACTOR
VAR_INPUT
END_VAR
VAR_OUTPUT
END_VAR
VAR
	{attribute 'instance-path'} 
    {attribute 'noinit'} 
	strInstancePath: STRING;
	strFullObjectPath: STRING;
	stEvent: ST_EVENT;
  stParams: ST_HMI_CYLINDER;
  stValve:  ST_HMI_VALVE;
	bAck: BOOL;
	itfOpMode:			I_OP_MODE;
	itfValveToBase:		I_BASE_VALVE;
	itfValveToWork: 	I_BASE_VALVE;
	itfSensorInBase: 	I_BINARY_SWITCH;
	itfSensorInWork: 	I_BINARY_SWITCH;
	
	tonToBase: Tc2_Standard.TON;
	tToBase: TIME;
	tonToWork: Tc2_Standard.TON;
	tToWork: TIME;
	bViewToBase: BOOL;
	bViewToWork: BOOL;
	//Locking
	bLockWorkMovement: BOOL:=FALSE;
	bLockBaseMovement: BOOL:=FALSE;
	bLockWorkActive: BOOL:=FALSE;
	bLockBaseActive: BOOL:=FALSE;
	strLockedByObject: STRING;
	
	bTestEvent: BOOL:=0;
	iStateInfo: INT;
END_VAR

METHOD FB_init : BOOL
VAR_INPUT
	bInitRetains : BOOL; // if TRUE, the retain variables are initialized (warm start / cold start)
	bInCopyCode : BOOL;  // if TRUE, the instance afterwards gets moved into the copy code (online change)
	itfOpMode:		I_OP_MODE;
	itfValveToBase: I_BASE_VALVE;
	itfValveToWork: I_BASE_VALVE;
	itfSensorInBase: I_BINARY_SWITCH;
	itfSensorInWork: I_BINARY_SWITCH;
	tTimeOutToBase: TIME;
	tTimeOutToWork: TIME;
END_VAR
THIS^.itfOpMode:=		itfOpMode;		
THIS^.itfValveToBase:=  itfValveToBase; 
THIS^.itfValveToWork:=  itfValveToWork; 
THIS^.itfSensorInBase:= itfSensorInBase;
THIS^.itfSensorInWork:= itfSensorInWork;
THIS^.tToBase:= 		tTimeOutToBase;
THIS^.tToWork:= 		tTimeOutToWork;
END_METHOD

{warning 'Methodenimplementierung hinzufügen'}
METHOD M_LockMovment
VAR_INPUT
	bLockBaseMovement	: BOOL;
	bLockWorkMovement	: BOOL;
	itfObject	: I_GENERAL_OBJECT;
END_VAR
THIS^.bLockBaseMovement:=	bLockBaseMovement;
THIS^.bLockWorkMovement:= 	bLockWorkMovement;
THIS^.strLockedByObject:= 	itfObject.P_FullObjectPath;
END_METHOD

METHOD M_Run
VAR

END_VAR
//Abarbeiten der geerbten Objekte
F_HandleInheritanceObjectInMRun(itfInheritanceObject:=THIS^.itfValveToBase,itfThisObject:=THIS^);
F_HandleInheritanceObjectInMRun(itfInheritanceObject:=THIS^.itfValveToWork,itfThisObject:=THIS^);
F_HandleInheritanceObjectInMRun(itfInheritanceObject:=THIS^.itfSensorInBase,itfThisObject:=THIS^);
F_HandleInheritanceObjectInMRun(itfInheritanceObject:=THIS^.itfValveToWork,itfThisObject:=THIS^);


//Handle Timeout Fault
IF TRUE 
AND (tonToBase.Q 
AND NOT stEvent.bEventActive 
AND 
(THIS^.itfOpMode.P_OP_MODE_STATE=OP_MODE.AUTO 
OR THIS^.itfOpMode.P_OP_MODE_STATE=OP_MODE.DEBUG 
OR THIS^.itfOpMode.P_OP_MODE_STATE=OP_MODE.INIT))
THEN
	stEvent.bEventActive:= TRUE;
	stEvent.enumEventType:= ENUM_EVENT_TYPE.Bl2_Message;
	stEvent.strEventText:= F_RET_TXTLIST_ENTRY(strPortNr:='851',strID:='2',strTxtLstName:='TXT_LIST_PNEMATIC_ACTOR');
	stEvent.strObject:= THIS^.P_FullObjectPath;
END_IF
IF (THIS^.tToBase=T#0MS) THEN
	stEvent.bEventActive:= FALSE;
END_IF


IF TRUE
AND (tonToWork.Q  
AND NOT stEvent.bEventActive 
AND 
(THIS^.itfOpMode.P_OP_MODE_STATE=OP_MODE.AUTO 
OR THIS^.itfOpMode.P_OP_MODE_STATE=OP_MODE.DEBUG 
OR THIS^.itfOpMode.P_OP_MODE_STATE=OP_MODE.INIT)) 
THEN
	stEvent.bEventActive:= TRUE;
	stEvent.enumEventType:= ENUM_EVENT_TYPE.Ye4_Stateinfo;
	stEvent.strEventText:= F_RET_TXTLIST_ENTRY(strPortNr:='851',strID:='1',strTxtLstName:='TXT_LIST_PNEMATIC_ACTOR');
	stEvent.strObject:= THIS^.P_FullObjectPath;
END_IF
IF (THIS^.tToWork=T#0MS) THEN
	stEvent.bEventActive:= FALSE;;
END_IF

//Event movment is locked
IF THIS^.bLockWorkActive OR THIS^.bLockBaseActive THEN
	stEvent.bEventActive:= TRUE;
	stEvent.enumEventType:= ENUM_EVENT_TYPE.Bl3_Hint;
	stEvent.strEventText:= F_RET_TXTLIST_ENTRY(strPortNr:='851',strID:='16',strTxtLstName:='TXT_LIST_PNEMATIC_ACTOR');
	stEvent.strEventText:= Tc2_Standard.CONCAT(stEvent.strEventText,' ');
	stEvent.strEventText:= Tc2_Standard.CONCAT(stEvent.strEventText,THIS^.strLockedByObject);
	stEvent.strObject:= THIS^.P_FullObjectPath;
	//No Timeout
	tonToBase.IN:= FALSE;
	tonToWork.IN:= FALSE;
END_IF



IF THIS^.P_Global_Ack (*AND (tonToBase.Q OR tonToWork.Q) *)THEN
	stEvent.bEventActive:= FALSE;
	tonToBase.IN:= FALSE;
	tonToWork.IN:= FALSE;
	THIS^.bLockWorkActive:=FALSE;
	THIS^.bLockBaseActive:=FALSE;
END_IF



IF THIS^.P_State=E_POS_STATE.InBasePos THEN
	tonToBase.IN:= FALSE;
END_IF
IF THIS^.P_State=E_POS_STATE.InWorkPos THEN
	tonTowork.IN:= FALSE;
END_IF

tonToWork(PT:=tToWork);
tonToBase(PT:=tToBase);
END_METHOD

{warning 'Methodenimplementierung hinzufügen'}
METHOD M_Stop
IF NOT THIS^.stEvent.bEventActive AND 
(THIS^.itfOpMode.P_OP_MODE_STATE=OP_MODE.AUTO 
OR THIS^.itfOpMode.P_OP_MODE_STATE=OP_MODE.INIT 
OR THIS^.itfOpMode.P_OP_MODE_STATE=OP_MODE.DEBUG
OR THIS^.itfOpMode.P_OP_MODE_STATE=OP_MODE.MANUAL)THEN
	THIS^.itfValveToBase.M_close();
	THIS^.itfValveToWork.M_Close();
	THIS^.tonToBase.IN:= FALSE;
	THIS^.tonToWork.IN:= FALSE;
END_IF
bViewToBase:= FALSE;
bViewToWork:= FALSE;
END_METHOD

{warning 'Methodenimplementierung hinzufügen'}
METHOD M_ToBasePos
IF (*NOT THIS^.stEvent.bEventActive AND*)
(THIS^.itfOpMode.P_OP_MODE_STATE=OP_MODE.AUTO 
OR THIS^.itfOpMode.P_OP_MODE_STATE=OP_MODE.INIT 
OR THIS^.itfOpMode.P_OP_MODE_STATE=OP_MODE.DEBUG
OR THIS^.itfOpMode.P_OP_MODE_STATE=OP_MODE.MANUAL) THEN
	IF NOT THIS^.bLockBaseMovement THEN
		THIS^.itfValveToBase.M_OPEN();
		THIS^.itfValveToWork.M_Close();
		THIS^.tonToBase.IN:= TRUE;
		THIS^.tonToWork.IN:= FALSE;
	ELSE
		THIS^.bLockBaseActive:=TRUE;
	END_IF;	
END_IF;

bViewToBase:= TRUE;
bViewToWork:= FALSE;
END_METHOD

{warning 'Methodenimplementierung hinzufügen'}
METHOD M_ToWorkPos
IF (*NOT THIS^.stEvent.bEventActive AND *)
(THIS^.itfOpMode.P_OP_MODE_STATE=OP_MODE.AUTO 
OR THIS^.itfOpMode.P_OP_MODE_STATE=OP_MODE.INIT 
OR THIS^.itfOpMode.P_OP_MODE_STATE=OP_MODE.DEBUG
OR THIS^.itfOpMode.P_OP_MODE_STATE=OP_MODE.MANUAL)THEN
	IF NOT THIS^.bLockWorkMovement THEN
		THIS^.itfValveToWork.M_OPEN();
		THIS^.itfValveToBase.M_Close();
		THIS^.tonToWork.IN:= TRUE;
		THIS^.tonToBase.IN:= FALSE;
	ELSE
		THIS^.bLockWorkActive:=TRUE;
	END_IF
END_IF
bViewToBase:= FALSE;
bViewToWork:= TRUE;
END_METHOD

{warning 'Methodenimplementierung hinzufügen'}
METHOD M_UnLockMovment
THIS^.bLockBaseMovement:=	FALSE;
THIS^.bLockWorkMovement:= 	false;
END_METHOD


PROPERTY P_Event : ST_EVENT
GET
VAR
	stEventTemp: ST_EVENT;
END_VAR
P_Event:= stEvent;
END_GET
SET
END_SET
END_PROPERTY


PROPERTY P_FullObjectPath : STRING
GET
P_FullObjectPath:= THIS^.strFullObjectPath;
END_GET
SET
THIS^.strFullObjectPath:= P_FullObjectPath;
END_SET
END_PROPERTY


PROPERTY P_Global_Ack : BOOL
GET
P_Global_Ack:= THIS^.bAck;
END_GET
SET
THIS^.bAck:=P_Global_Ack;
END_SET
END_PROPERTY


PROPERTY P_GlobalID : STRING
GET
P_GlobalID:= THIS^.strInstancePath;
END_GET
END_PROPERTY


PROPERTY P_State : E_POS_STATE
GET
P_State:=E_POS_STATE.NoDefPos;

//Actor in BasePos
IF THIS^.itfSensorInBase.P_Active THEN
	P_State:=E_POS_STATE.InBasePos;
ELSE;
END_IF

//Actor in WorkPos
IF THIS^.itfSensorInWork.P_Active THEN
	P_State:=E_POS_STATE.InWorkPos;
ELSE;
END_IF

//Actor in BasePos
IF THIS^.itfSensorInBase.P_Active AND THIS^.itfValveToBase.P_IS_OPEN THEN
	P_State:=E_POS_STATE.InBasePos;
ELSE;
END_IF

//Actor in WorkPos
IF THIS^.itfSensorInWork.P_Active AND THIS^.itfValveToWork.P_IS_OPEN THEN
	P_State:=E_POS_STATE.InWorkPos;
ELSE;
END_IF

IF  NOT THIS^.itfSensorInWork.P_Active AND NOT THIS^.itfSensorInBase.P_Active THEN
	P_State:=E_POS_STATE.NoDefPos;
	//Actor Move to Base
	IF THIS^.itfValveToBase.P_IS_OPEN AND THIS^.itfValveToWork.P_IS_CLOSE THEN
		P_State:= E_POS_STATE.MoveToBase;
	ELSE;	
	END_IF
	//Actor Move to Work
	IF THIS^.itfValveToWork.P_IS_OPEN AND THIS^.itfValveToBase.P_IS_CLOSE THEN
		P_State:= E_POS_STATE.MoveToWork;
	ELSE;	
	END_IF	
ELSE;
END_IF
IF  THIS^.itfSensorInWork.P_Active AND THIS^.itfSensorInBase.P_Active THEN
	P_State:=E_POS_STATE.NoDefPos;
END_IF

IF THIS^.bLockBaseActive THEN
	P_State:=E_POS_STATE.MoveToBaseLock;
END_IF

IF THIS^.bLockWorkActive THEN
	P_State:=E_POS_STATE.MoveToWorkLock;
END_IF

 CASE P_State OF
	E_POS_STATE.InBasePos: 			THIS^.iStateInfo:=0;
	E_POS_STATE.InWorkPos:			THIS^.iStateInfo:=1;
	E_POS_STATE.InMidPos:			THIS^.iStateInfo:=2;
	E_POS_STATE.InBasePosValveOff:	THIS^.iStateInfo:=3;
	E_POS_STATE.InWorkPosValveOff:	THIS^.iStateInfo:=4;
	E_POS_STATE.NoDefPos:			THIS^.iStateInfo:=5;
	E_POS_STATE.MoveToBase:			THIS^.iStateInfo:=6;
	E_POS_STATE.MoveToWork:			THIS^.iStateInfo:=7;
	E_POS_STATE.TimeOutToWork:		THIS^.iStateInfo:=8;
	E_POS_STATE.TimeOutToBase:		THIS^.iStateInfo:=9;
	E_POS_STATE.MoveToBaseLock:		THIS^.iStateInfo:=10;
	E_POS_STATE.MoveToWorkLock:		THIS^.iStateInfo:=11;
	ELSE
		iStateInfo:=99;
 END_CASE
END_GET
END_PROPERTY


PROPERTY P_TimeOutToBase : TIME
GET
P_TimeOutToBase:= tonToBase.PT;
END_GET
SET
tToBase:= P_TimeOutToBase;
END_SET
END_PROPERTY


PROPERTY P_TimeOutToWork : TIME
GET
P_TimeOutToWork:= tonToWork.PT;
END_GET
SET
tToWork:= P_TimeOutToWork;
END_SET
END_PROPERTY

END_FUNCTION_BLOCK

// ---- MODULE/ACTOR_VALVE/PNEUMATIC_ACTOR/POU/FB_ZYLINDER_TWO_WAY_MID_POS.TcPOU
{attribute 'reflection'} 
{attribute 'no_explicit_call' := 'do not call this POU directly'} 
FUNCTION_BLOCK FB_ZYLINDER_TWO_WAY_MID_POS IMPLEMENTS I_PNEU_ACTOR
VAR_INPUT
END_VAR
VAR_OUTPUT
END_VAR
VAR
	{attribute 'instance-path'} 
    {attribute 'noinit'} 
	strInstancePath: STRING;
	strFullObjectPath: STRING;
	stEvent: ST_EVENT;
	bAck: BOOL;
	itfOpMode:			I_OP_MODE;
	itfValveToBase:		I_BASE_VALVE;
	itfValveToWork: 	I_BASE_VALVE;
	itfSensorInBase: 	I_BINARY_SWITCH;
	itfSensorInWork: 	I_BINARY_SWITCH;
	itfSensorInMid: 	I_BINARY_SWITCH;
	tDebounceTimeMid: TIME;
	tonDebounceTimeMid:		Tc2_Standard.TON;
	tonToBase: Tc2_Standard.TON;
	tToBase: TIME;
	tonToWork: Tc2_Standard.TON;
	tToWork: TIME;
	bViewToBase: BOOL;
	bViewToWork: BOOL;
		//Locking
	bLockWorkMovement: BOOL:=FALSE;
	bLockBaseMovement: BOOL:=FALSE;
	bLockWorkActive: BOOL:=FALSE;
	bLockBaseActive: BOOL:=FALSE;
	strLockedByObject: STRING;
	
END_VAR

METHOD FB_init : BOOL
VAR_INPUT
	bInitRetains : BOOL; // if TRUE, the retain variables are initialized (warm start / cold start)
	bInCopyCode : BOOL;  // if TRUE, the instance afterwards gets moved into the copy code (online change)
	itfOpMode:		I_OP_MODE;
	itfValveToBase: I_BASE_VALVE;
	itfValveToWork: I_BASE_VALVE;
	itfSensorInBase: I_BINARY_SWITCH;
	itfSensorInWork: I_BINARY_SWITCH;
	itfSensorInMid: I_BINARY_SWITCH;
	tTimeOutToBase: TIME;
	tTimeOutToWork: TIME;
	tDebounceTimeMid: TIME;
END_VAR
THIS^.itfOpMode:=		itfOpMode;		
THIS^.itfValveToBase:=  itfValveToBase; 
THIS^.itfValveToWork:=  itfValveToWork; 
THIS^.itfSensorInBase:= itfSensorInBase;
THIS^.itfSensorInWork:= itfSensorInWork;
THIS^.itfSensorInMid:=	itfSensorInMid;
THIS^.tToBase:= 		tTimeOutToBase;
THIS^.tToWork:= 		tTimeOutToWork;
THIS^.tDebounceTimeMid:=tDebounceTimeMid;
END_METHOD

{warning 'Methodenimplementierung hinzufügen'}
METHOD M_LockMovment
VAR_INPUT
	bLockBaseMovement	: BOOL;
	bLockWorkMovement	: BOOL;
	itfObject	: I_GENERAL_OBJECT;
END_VAR
THIS^.bLockBaseMovement:=	bLockBaseMovement;
THIS^.bLockWorkMovement:= 	bLockWorkMovement;
THIS^.strLockedByObject:= 	itfObject.P_FullObjectPath;
END_METHOD

METHOD M_Run
VAR

END_VAR
//Abarbeiten der geerbten Objekte
F_HandleInheritanceObjectInMRun(itfInheritanceObject:=THIS^.itfValveToBase,itfThisObject:=THIS^);
F_HandleInheritanceObjectInMRun(itfInheritanceObject:=THIS^.itfValveToWork,itfThisObject:=THIS^);
F_HandleInheritanceObjectInMRun(itfInheritanceObject:=THIS^.itfSensorInBase,itfThisObject:=THIS^);
F_HandleInheritanceObjectInMRun(itfInheritanceObject:=THIS^.itfSensorInWork,itfThisObject:=THIS^);
F_HandleInheritanceObjectInMRun(itfInheritanceObject:=THIS^.itfSensorInMid,itfThisObject:=THIS^);




//Handle Timeout Fault
IF tonToBase.Q AND NOT stEvent.bEventActive AND (THIS^.itfOpMode.P_OP_MODE_STATE=OP_MODE.AUTO OR THIS^.itfOpMode.P_OP_MODE_STATE=OP_MODE.DEBUG OR THIS^.itfOpMode.P_OP_MODE_STATE=OP_MODE.INIT) THEN
	stEvent.bEventActive:= TRUE;
	stEvent.enumEventType:= ENUM_EVENT_TYPE.Bl2_Message;
	stEvent.strEventText:= F_RET_TXTLIST_ENTRY(strPortNr:='851',strID:='2',strTxtLstName:='TXT_LIST_PNEMATIC_ACTOR');
	stEvent.strObject:= THIS^.P_FullObjectPath;
END_IF

IF tonToWork.Q  AND NOT stEvent.bEventActive AND (THIS^.itfOpMode.P_OP_MODE_STATE=OP_MODE.AUTO OR THIS^.itfOpMode.P_OP_MODE_STATE=OP_MODE.DEBUG OR THIS^.itfOpMode.P_OP_MODE_STATE=OP_MODE.INIT) THEN
	stEvent.bEventActive:= TRUE;
	stEvent.enumEventType:= ENUM_EVENT_TYPE.Ye4_Stateinfo;
	stEvent.strEventText:= F_RET_TXTLIST_ENTRY(strPortNr:='851',strID:='1',strTxtLstName:='TXT_LIST_PNEMATIC_ACTOR');
	stEvent.strObject:= THIS^.P_FullObjectPath;
END_IF

//Event movment is locked
IF THIS^.bLockWorkActive OR THIS^.bLockBaseActive THEN
	stEvent.bEventActive:= TRUE;
	stEvent.enumEventType:= ENUM_EVENT_TYPE.Ye4_Stateinfo;
	stEvent.strEventText:= F_RET_TXTLIST_ENTRY(strPortNr:='851',strID:='16',strTxtLstName:='TXT_LIST_PNEMATIC_ACTOR');
	stEvent.strEventText:= Tc2_Standard.CONCAT(stEvent.strEventText,' ');
	stEvent.strEventText:= Tc2_Standard.CONCAT(stEvent.strEventText,THIS^.strLockedByObject);
	stEvent.strObject:= THIS^.P_FullObjectPath;
END_IF

IF THIS^.P_Global_Ack (*AND (tonToBase.Q OR tonToWork.Q) *)THEN
	stEvent.bEventActive:= FALSE;
	tonToBase.IN:= FALSE;
	tonToWork.IN:= FALSE;
	THIS^.bLockWorkActive:=FALSE;
	THIS^.bLockBaseActive:=FALSE;
END_IF



IF THIS^.P_State=E_POS_STATE.InBasePos OR P_State=E_POS_STATE.InMidPos THEN
	tonToBase.IN:= FALSE;
END_IF
IF THIS^.P_State=E_POS_STATE.InWorkPos OR P_State=E_POS_STATE.InMidPos THEN
	tonTowork.IN:= FALSE;
END_IF

tonToWork(PT:=tToWork);
tonToBase(PT:=tToBase);

tonDebounceTimeMid.IN:=THIS^.itfSensorInMid.P_Active;
tonDebounceTimeMid(PT:=tDebounceTimeMid);
END_METHOD

{warning 'Methodenimplementierung hinzufügen'}
METHOD M_Stop
IF NOT THIS^.stEvent.bEventActive AND 
(THIS^.itfOpMode.P_OP_MODE_STATE=OP_MODE.AUTO 
OR THIS^.itfOpMode.P_OP_MODE_STATE=OP_MODE.INIT 
OR THIS^.itfOpMode.P_OP_MODE_STATE=OP_MODE.DEBUG
OR THIS^.itfOpMode.P_OP_MODE_STATE=OP_MODE.MANUAL)THEN
	THIS^.itfValveToBase.M_close();
	THIS^.itfValveToWork.M_Close();
	THIS^.tonToBase.IN:= FALSE;
	THIS^.tonToWork.IN:= FALSE;
END_IF
bViewToBase:= FALSE;
bViewToWork:= FALSE;
END_METHOD

{warning 'Methodenimplementierung hinzufügen'}
METHOD M_ToBasePos
IF NOT THIS^.stEvent.bEventActive
AND (THIS^.itfOpMode.P_OP_MODE_STATE=OP_MODE.AUTO 
OR THIS^.itfOpMode.P_OP_MODE_STATE=OP_MODE.INIT 
OR THIS^.itfOpMode.P_OP_MODE_STATE=OP_MODE.DEBUG
OR THIS^.itfOpMode.P_OP_MODE_STATE=OP_MODE.MANUAL) THEN
	IF NOT THIS^.bLockBaseMovement THEN
		THIS^.itfValveToBase.M_OPEN();
		THIS^.itfValveToWork.M_Close();
		THIS^.tonToBase.IN:= TRUE;
		THIS^.tonToWork.IN:= FALSE;
	ELSE
		THIS^.bLockBaseActive:=TRUE;
	END_IF
END_IF;

bViewToBase:= TRUE;
bViewToWork:= FALSE;
END_METHOD

{warning 'Methodenimplementierung hinzufügen'}
METHOD M_ToWorkPos
IF NOT THIS^.stEvent.bEventActive AND 
(THIS^.itfOpMode.P_OP_MODE_STATE=OP_MODE.AUTO 
OR THIS^.itfOpMode.P_OP_MODE_STATE=OP_MODE.INIT 
OR THIS^.itfOpMode.P_OP_MODE_STATE=OP_MODE.DEBUG
OR THIS^.itfOpMode.P_OP_MODE_STATE=OP_MODE.MANUAL)THEN
	IF NOT THIS^.bLockWorkMovement THEN
		THIS^.itfValveToWork.M_OPEN();
		THIS^.itfValveToBase.M_Close();
		THIS^.tonToWork.IN:= TRUE;
		THIS^.tonToBase.IN:= FALSE;
	ELSE
		THIS^.bLockWorkActive:=TRUE;
	END_IF	
END_IF
bViewToBase:= FALSE;
bViewToWork:= TRUE;
END_METHOD

{warning 'Methodenimplementierung hinzufügen'}
METHOD M_UnLockMovment
THIS^.bLockBaseMovement:=	FALSE;
THIS^.bLockWorkMovement:= 	false;
END_METHOD


PROPERTY P_Event : ST_EVENT
GET
VAR
	stEventTemp: ST_EVENT;
END_VAR
P_Event:= stEvent;
END_GET
SET
END_SET
END_PROPERTY


PROPERTY P_FullObjectPath : STRING
GET
P_FullObjectPath:= THIS^.strFullObjectPath;
END_GET
SET
THIS^.strFullObjectPath:= P_FullObjectPath;
END_SET
END_PROPERTY


PROPERTY P_Global_Ack : BOOL
GET
P_Global_Ack:= THIS^.bAck;
END_GET
SET
THIS^.bAck:=P_Global_Ack;
END_SET
END_PROPERTY


PROPERTY P_GlobalID : STRING
GET
P_GlobalID:= THIS^.strInstancePath;
END_GET
END_PROPERTY


PROPERTY P_State : E_POS_STATE
GET
P_State:=E_POS_STATE.NoDefPos;

//Actor in BasePos
IF THIS^.itfSensorInBase.P_Active THEN
	P_State:=E_POS_STATE.InBasePos;
ELSE;
END_IF

//Actor in WorkPos
IF THIS^.itfSensorInWork.P_Active THEN
	P_State:=E_POS_STATE.InWorkPos;
ELSE;
END_IF

//Actor in MidPos
IF THIS^.tonDebounceTimeMid.Q THEN
	P_State:=E_POS_STATE.InMidPos;
ELSE;
END_IF

//Actor in BasePos
IF THIS^.itfSensorInBase.P_Active AND THIS^.itfValveToBase.P_IS_OPEN THEN
	P_State:=E_POS_STATE.InBasePos;
ELSE;
END_IF

//Actor in WorkPos
IF THIS^.itfSensorInWork.P_Active AND THIS^.itfValveToWork.P_IS_OPEN THEN
	P_State:=E_POS_STATE.InWorkPos;
ELSE;
END_IF

IF  NOT THIS^.itfSensorInWork.P_Active AND NOT THIS^.itfSensorInBase.P_Active AND NOT THIS^.tonDebounceTimeMid.Q THEN
	P_State:=E_POS_STATE.NoDefPos;
	//Actor Move to Base
	IF THIS^.itfValveToBase.P_IS_OPEN AND THIS^.itfValveToWork.P_IS_CLOSE THEN
		P_State:= E_POS_STATE.MoveToBase;
	ELSE;	
	END_IF
	//Actor Move to Work
	IF THIS^.itfValveToWork.P_IS_OPEN AND THIS^.itfValveToBase.P_IS_CLOSE THEN
		P_State:= E_POS_STATE.MoveToWork;
	ELSE;	
	END_IF	
ELSE;
END_IF
IF  THIS^.itfSensorInWork.P_Active AND THIS^.itfSensorInBase.P_Active THEN
	P_State:=E_POS_STATE.NoDefPos;
END_IF

IF THIS^.bLockBaseActive THEN
	P_State:=E_POS_STATE.MoveToBaseLock;
END_IF

IF THIS^.bLockWorkActive THEN
	P_State:=E_POS_STATE.MoveToWorkLock;
END_IF
END_GET
END_PROPERTY


PROPERTY P_TimeOutToBase : TIME
GET
P_TimeOutToBase:= tonToBase.PT;
END_GET
SET
tToBase:= P_TimeOutToBase;
END_SET
END_PROPERTY


PROPERTY P_TimeOutToWork : TIME
GET
P_TimeOutToWork:= tonToWork.PT;
END_GET
SET
tToWork:= P_TimeOutToWork;
END_SET
END_PROPERTY

END_FUNCTION_BLOCK

// ---- MODULE/BUS_DIAG/POU/FB_EC_MASTER.TcPOU
{attribute 'reflection'} 
{attribute 'no_explicit_call' := 'do not call this POU directly'} 
FUNCTION_BLOCK FB_EC_MASTER IMPLEMENTS I_Master
VAR_INPUT
END_VAR
VAR_OUTPUT
END_VAR
VAR
	
	{attribute 'instance-path'} 
    {attribute 'noinit'} 
	strInstancePath: STRING;
	strFullObjectPath: STRING;
	stEvent: ST_EVENT;
	bAck: BOOL;
	
	uiDevState AT %I*: 	UINT;
	uiLastDevState: 	UINT;
	
	itfLogEvents: 		I_HANDLE_EVENTS;
	fbEventState: 		FB_CREATE_EVENT(itfLogEvents:= itfLogEvents, itfID:=THIS^);
	bAnyEvent:			BOOL;
END_VAR

METHOD FB_init : BOOL
VAR_INPUT
	bInitRetains : BOOL; // if TRUE, the retain variables are initialized (warm start / cold start)
	bInCopyCode : BOOL;  // if TRUE, the instance afterwards gets moved into the copy code (online change)
	itfLogEvents: 		I_HANDLE_EVENTS;
END_VAR
this^.itfLogEvents:=itfLogEvents;
END_METHOD


(*=== Method: M_Run  ============================================

 @brief: Here is the global code (Timer, Event, Flange,...)*)
METHOD M_Run
VAR
strTemp: STRING;	
END_VAR
//Get own Name
THIS^.strFullObjectPath:= F_RET_TXTLIST_ENTRY(strPortNr:='851', strID:=THIS^.strInstancePath, strTxtLstName:='TXT_LIST_OBJECTS');
bAnyEvent:=FALSE;

//0x0001 = Link error
strTemp:= Tc2_Standard.CONCAT(THIS^.strFullObjectPath, ' -> ');
strTemp:=Tc2_Standard.CONCAT(strTemp, 'Link error');
IF THIS^.uiDevState = 16#0001 THEN
	THIS^.fbEventState.M_Log(strTemp,enum_event_type.Ye4_Stateinfo,THIS^.itfLogEvents);
	bAnyEvent:=TRUE;
END_IF
//0x0002 = I/O locked after link error (I/O reset required)
strTemp:= Tc2_Standard.CONCAT(THIS^.strFullObjectPath, ' -> ');
strTemp:=Tc2_Standard.CONCAT(strTemp, 'I/O locked after link error (I/O reset required)');
IF THIS^.uiDevState = 16#0002 THEN
	THIS^.fbEventState.M_Log(strTemp,enum_event_type.Ye4_Stateinfo,THIS^.itfLogEvents);
	bAnyEvent:=TRUE;
END_IF
//0x0004 = Link error (redundancy adapter)
strTemp:= Tc2_Standard.CONCAT(THIS^.strFullObjectPath, ' -> ');
strTemp:=Tc2_Standard.CONCAT(strTemp, 'Link error (redundancy adapter)');
IF THIS^.uiDevState = 16#0004 THEN
	THIS^.fbEventState.M_Log(strTemp,enum_event_type.Ye4_Stateinfo,THIS^.itfLogEvents);
	bAnyEvent:=TRUE;
END_IF
//0x0008 = Missing one frame (redundancy mode)
strTemp:= Tc2_Standard.CONCAT(THIS^.strFullObjectPath, ' -> ');
strTemp:=Tc2_Standard.CONCAT(strTemp, 'Missing one frame (redundancy mode)');
IF THIS^.uiDevState = 16#0008 THEN
	THIS^.fbEventState.M_Log(strTemp,enum_event_type.Ye4_Stateinfo,THIS^.itfLogEvents);
	bAnyEvent:=TRUE;
END_IF
//0x0010 = Out of send resources (I/O reset required)
strTemp:= Tc2_Standard.CONCAT(THIS^.strFullObjectPath, ' -> ');
strTemp:=Tc2_Standard.CONCAT(strTemp, 'Out of send resources (I/O reset required)');
IF THIS^.uiDevState = 16#0010 THEN
	THIS^.fbEventState.M_Log(strTemp,enum_event_type.Ye4_Stateinfo,THIS^.itfLogEvents);
	bAnyEvent:=TRUE;
END_IF
//0x0020 = Watchdog triggered
strTemp:= Tc2_Standard.CONCAT(THIS^.strFullObjectPath, ' -> ');
strTemp:=Tc2_Standard.CONCAT(strTemp, 'Watchdog triggered');
IF THIS^.uiDevState = 16#0020 THEN
	THIS^.fbEventState.M_Log(strTemp,enum_event_type.Ye4_Stateinfo,THIS^.itfLogEvents);
	bAnyEvent:=TRUE;
END_IF
//0x0040 = Ethernet driver (miniport) not found
strTemp:= Tc2_Standard.CONCAT(THIS^.strFullObjectPath, ' -> ');
strTemp:=Tc2_Standard.CONCAT(strTemp, 'Ethernet driver (miniport) not found');
IF THIS^.uiDevState = 16#0040 THEN
	THIS^.fbEventState.M_Log(strTemp,enum_event_type.Ye4_Stateinfo,THIS^.itfLogEvents);
	bAnyEvent:=TRUE;
END_IF
//0x0080 = I/O reset active
strTemp:= Tc2_Standard.CONCAT(THIS^.strFullObjectPath, ' -> ');
strTemp:=Tc2_Standard.CONCAT(strTemp, 'I/O reset active');
IF THIS^.uiDevState = 16#0080 THEN
	THIS^.fbEventState.M_Log(strTemp,enum_event_type.Ye4_Stateinfo,THIS^.itfLogEvents);
	bAnyEvent:=TRUE;
END_IF
//0x0100 = At least one device in 'INIT' state
strTemp:= Tc2_Standard.CONCAT(THIS^.strFullObjectPath, ' -> ');
strTemp:=Tc2_Standard.CONCAT(strTemp, 'At least one device in "INIT" state');
IF THIS^.uiDevState = 16#0100 THEN
	THIS^.fbEventState.M_Log(strTemp,enum_event_type.Ye4_Stateinfo,THIS^.itfLogEvents);
	bAnyEvent:=TRUE;
END_IF
//0x0200 = At least one device in 'PRE-OP' state
strTemp:= Tc2_Standard.CONCAT(THIS^.strFullObjectPath, ' -> ');
strTemp:=Tc2_Standard.CONCAT(strTemp, 'At least one device in "PRE-OP" state');
IF THIS^.uiDevState = 16#0200 THEN
	THIS^.fbEventState.M_Log(strTemp,enum_event_type.Ye4_Stateinfo,THIS^.itfLogEvents);
	bAnyEvent:=TRUE;
END_IF
//0x0400 = At least one device in 'SAFE-OP' state
strTemp:= Tc2_Standard.CONCAT(THIS^.strFullObjectPath, ' -> ');
strTemp:=Tc2_Standard.CONCAT(strTemp, 'At least one device in "SAFE-OP" state');
IF THIS^.uiDevState = 16#0400 THEN
	THIS^.fbEventState.M_Log(strTemp,enum_event_type.Ye4_Stateinfo,THIS^.itfLogEvents);
	bAnyEvent:=TRUE;
END_IF
//0x0800 = At least one device indicates an error state
strTemp:= Tc2_Standard.CONCAT(THIS^.strFullObjectPath, ' -> ');
strTemp:=Tc2_Standard.CONCAT(strTemp, 'At least one device indicates an error stat');
IF THIS^.uiDevState = 16#0800 THEN
	THIS^.fbEventState.M_Log(strTemp,enum_event_type.Ye4_Stateinfo,THIS^.itfLogEvents);
	bAnyEvent:=TRUE;
END_IF
//0x1000 = DC not in sync
strTemp:= Tc2_Standard.CONCAT(THIS^.strFullObjectPath, ' -> ');
strTemp:=Tc2_Standard.CONCAT(strTemp, 'DC not in sync');
IF THIS^.uiDevState = 16#1000 THEN
	THIS^.fbEventState.M_Log(strTemp,enum_event_type.Ye4_Stateinfo,THIS^.itfLogEvents);
	bAnyEvent:=TRUE;
END_IF




IF THIS^.uiDevState <= 0 
OR THIS^.bAck 
OR NOT bAnyEvent 
OR THIS^.uiLastDevState <>THIS^.uiDevState 
THEN	
	THIS^.fbEventState.M_Log('',enum_event_type.Gn0_None,THIS^.itfLogEvents);
	THIS^.fbEventState.M_Quit();
END_IF
THIS^.uiLastDevState:=THIS^.uiDevState;
END_METHOD

(*=== Property: P_Event  ============================================

 @param [set]: 	Set the Structure "ST_EVENT" from another Object
 @param [get]: 	Return the Structure "ST_EVENT", it contains the actual 
					event of the Object *)
PROPERTY P_Event : GenLib.ST_EVENT
GET
P_Event:= THIS^.stEvent;
END_GET
SET
THIS^.stEvent:=P_Event;
END_SET
END_PROPERTY

(*=== Property: P_FullObjectPath  ============================================

 @param [set]: 	Set the Object Path (Clear String of Object)
 @param [get]: 	Return the Objectpath *)
PROPERTY P_FullObjectPath : STRING
GET
P_FullObjectPath:= THIS^.strFullObjectPath;
END_GET
SET
THIS^.strFullObjectPath:=P_FullObjectPath;
END_SET
END_PROPERTY

(*=== Property: P_Global_Ack  ============================================

 @param [set]: 	Set the Bit for Ack from another Object
 @param [get]: 	Return the state of Ack Bit*)
PROPERTY P_Global_Ack : BOOL
GET
P_Global_Ack:= bAck;
END_GET
SET
bAck:=P_Global_Ack;
END_SET
END_PROPERTY

(*=== Property: P_GlobalID  ============================================

 @param [set]: 	-
 @param [get]: 	Return the string of instance path*)
PROPERTY P_GlobalID : STRING
GET
P_GlobalID:= THIS^.strInstancePath;
END_GET
END_PROPERTY

PROPERTY P_STATE : INT
GET
P_STATE:=UINT_TO_INT(this^.uiDevState);
END_GET
END_PROPERTY

END_FUNCTION_BLOCK

// ---- MODULE/BUS_DIAG/POU/FB_VISU_BUS_DIAG.TcPOU
FUNCTION_BLOCK FB_VISU_BUS_DIAG
VAR_INPUT
END_VAR
VAR_OUTPUT
END_VAR
VAR
	itfMaster:I_Master;
	xType: WORD; 		//16#00: Ethercat; 16#01Profinet; 
	strType: STRING;
	strName: STRING;
	dwColor: DWORD;
	dwColorFrame: DWORD;
	strState: STRING;
END_VAR

strName:=concat('',itfMaster.P_FullObjectPath);

CASE xType OF
16#00://Ethercat
	dwColorFrame:=color.dwYellow;
	strType:='Ethercat Master';
	CASE itfMaster.P_STATE OF
	16#0001:  strState:= 'Link error'										;dwColor:=color.dwRed;
	16#0002:  strState:= 'I/O locked after link error (I/O reset required)' ;dwColor:=color.dwRed;
	16#0004:  strState:= 'Link error (redundancy adapter)'                  ;dwColor:=color.dwRed;
	16#0008:  strState:= 'Missing one frame (redundancy mode)'              ;dwColor:=color.dwRed;
	16#0010:  strState:= 'Out of send resources (I/O reset required)'       ;dwColor:=color.dwRed;
	16#0020:  strState:= 'Watchdog triggered'                               ;dwColor:=color.dwRed;
	16#0040:  strState:= 'Ethernet driver (miniport) not found'             ;dwColor:=color.dwRed;
	16#0080:  strState:= 'I/O reset active'                                 ;dwColor:=color.dwRed;
	16#0100:  strState:= 'At least one device in "INIT" state'              ;dwColor:=color.dwRed;
	16#0200:  strState:= 'At least one device in "PRE-OP" state'            ;dwColor:=color.dwRed;
	16#0400:  strState:= 'At least one device in "SAFE-OP" state'           ;dwColor:=color.dwRed;
	16#0800:  strState:= 'At least one device indicates an error state'     ;dwColor:=color.dwRed;
	16#1000:  strState:= 'DC not in sync'                                   ;dwColor:=color.dwRed;
	ELSE	  strState:= 'OK'                                 				;dwColor:=color.dwGreen;
	END_CASE
	;
16#01:;//Profinet	
	dwColorFrame:=color.dwGreen;
	strType:='Profinet Master';
	CASE itfMaster.P_STATE OF
	//16#0001:  strState:= 'No link AT port 1'								;dwColorFrame:=color.dwRed;
	//16#0002:  strState:= 'No link AT port 2'                              ;dwColorFrame:=color.dwRed;
	16#0010:  strState:= 'Out of send resources (I/O reset required)'       ;dwColor:=color.dwRed;
	16#0080:  strState:= 'I/O reset active'                                 ;dwColor:=color.dwRed;
	ELSE	  strState:= 'OK'                                 				;dwColor:=color.dwGreen;
	END_CASE
END_CASE

METHOD FB_init : BOOL
VAR_INPUT
	bInitRetains : BOOL; // if TRUE, the retain variables are initialized (warm start / cold start)
	bInCopyCode : BOOL;  // if TRUE, the instance afterwards gets moved into the copy code (online change)
	itfMaster:I_Master;
	xType: WORD; 		//16#00: Ethercat; 16#01Profinet; 
END_VAR
THIS^.itfMaster:=itfMaster;
this^.xType:=xType;
END_METHOD

END_FUNCTION_BLOCK

// ---- MODULE/BYTES_TO_WORD/POU/FB_BYTES_TO_WORD.TcPOU
FUNCTION_BLOCK FB_BYTES_TO_WORD IMPLEMENTS I_ANALOG_IN
VAR_INPUT
END_VAR
VAR_OUTPUT
END_VAR
VAR


uBytestoWord:					U_BytesToWord;
//Für Input
	bBytesIn1					AT %I* :BYTE;
	bBytesIn2					AT %I* :BYTE;
	wWordOut:					WORD;		

	i:							INT;
	


END_VAR

(*=== Method: M_Run  ============================================

 @brief: Here is the global code (Timer, Event, Flange,...)*)
METHOD M_Run
i:=i+1;
//Eingangsdaten Wandeln
uBytestoWord.arByteIn[0]:=bBytesIn2;
uBytestoWord.arByteIn[1]:=bBytesIn1;
wWordOut:=uBytestoWord.uintOut;
END_METHOD

(*=== Property: P_Event  ============================================

 @param [set]: 	Set the Structure "ST_EVENT" from another Object
 @param [get]: 	Return the Structure "ST_EVENT", it contains the actual 
					event of the Object *)
PROPERTY P_Event : GenLib.ST_EVENT
GET
END_GET
SET
END_SET
END_PROPERTY

{warning 'Eigenschaftenimplementierung hinzufügen'}
(*=== Property: P_FullObjectPath  ============================================

 @param [set]: 	Set the Object Path (Clear String of Object)
 @param [get]: 	Return the Objectpath *)
PROPERTY P_FullObjectPath : STRING
GET
END_GET
SET
END_SET
END_PROPERTY

{warning 'Eigenschaftenimplementierung hinzufügen'}
(*=== Property: P_Global_Ack  ============================================

 @param [set]: 	Set the Bit for Ack from another Object
 @param [get]: 	Return the state of Ack Bit*)
PROPERTY P_Global_Ack : BOOL
GET
END_GET
SET
END_SET
END_PROPERTY

{warning 'Eigenschaftenimplementierung hinzufügen'}
(*=== Property: P_GlobalID  ============================================

 @param [set]: 	-
 @param [get]: 	Return the string of instance path*)
PROPERTY P_GlobalID : STRING
GET
END_GET
END_PROPERTY

{warning 'Eigenschaftenimplementierung hinzufügen'}
PROPERTY P_Value : LREAL
GET
P_VALUE:= WORD_TO_LREAL(THIS^.wWordOut);
END_GET
END_PROPERTY

END_FUNCTION_BLOCK

// ---- MODULE/BYTES_TO_WORD/POU/FB_WORD_TO_BYTES.TcPOU
FUNCTION_BLOCK FB_WORD_TO_BYTES IMPLEMENTS I_WORD_TO_BYTES
VAR_INPUT
END_VAR
VAR_OUTPUT
END_VAR
VAR
	uWordToBytes:				U_BytesToWord ;
//Für Input
	bBytesOut1					AT %Q* :BYTE;
	bBytesOut2					AT %Q* :BYTE;
	lrWordIn:					LREAL;	
	
	lrUnscaledIn:				LREAL;
	lrScaledIn:					LREAL;
	temp_gain:					LREAL;
	temp_offset:				LREAL;
	lrX_Max:					LREAL	:=1;
	lrX_Min:					LREAL;
	lrY_Max:					LREAL	:=1;
	lrY_Min:					LREAL;	
	i:							INT;
END_VAR

METHOD FB_init : BOOL
VAR_INPUT
	bInitRetains : 				BOOL; // if TRUE, the retain variables are initialized (warm start / cold start)
	bInCopyCode : 				BOOL;  // if TRUE, the instance afterwards gets moved into the copy code (online change)
END_VAR
END_METHOD

(*=== Method: M_Run  ============================================

 @brief: Here is the global code (Timer, Event, Flange,...)*)
METHOD M_Run

VAR
END_VAR
i:=i+1;

uWordToBytes.uintOut:=LREAL_TO_WORD(lrWordIn);
bBytesOut2:=uWordToBytes.arByteIn[0];
bBytesOut1:=uWordToBytes.arByteIn[1];

IF lrY_Max = 0 THEN
	lrY_Max:=1;
END_IF
IF lrX_Max =0 THEN
	lrX_Max:=1;
END_IF

// Ausgang Scallieren
temp_gain := (lrY_Max - lrY_Min) / (lrX_Max - lrX_Min);
temp_offset := lrY_Min - lrX_Min * temp_gain;
lrWordIn := lrUnscaledIn * temp_gain + temp_offset;

IF lrUnscaledIn > lrX_Max THEN
    lrWordIn := REAL_TO_INT(lrY_Max);
ELSIF lrUnscaledIn < lrX_Min THEN
    lrWordIn := REAL_TO_INT(lrY_Min);
END_IF;
END_METHOD

(*=== Property: P_Event  ============================================

 @param [set]: 	Set the Structure "ST_EVENT" from another Object
 @param [get]: 	Return the Structure "ST_EVENT", it contains the actual 
					event of the Object *)
PROPERTY P_Event : GenLib.ST_EVENT
GET
END_GET
SET
END_SET
END_PROPERTY

(*=== Property: P_FullObjectPath  ============================================

 @param [set]: 	Set the Object Path (Clear String of Object)
 @param [get]: 	Return the Objectpath *)
PROPERTY P_FullObjectPath : STRING
GET
END_GET
SET
END_SET
END_PROPERTY

(*=== Property: P_Global_Ack  ============================================

 @param [set]: 	Set the Bit for Ack from another Object
 @param [get]: 	Return the state of Ack Bit*)
PROPERTY P_Global_Ack : BOOL
GET
END_GET
SET
END_SET
END_PROPERTY

(*=== Property: P_GlobalID  ============================================

 @param [set]: 	-
 @param [get]: 	Return the string of instance path*)
PROPERTY P_GlobalID : STRING
GET
END_GET
END_PROPERTY

PROPERTY P_VALUE : LREAL
GET
P_VALUE:=lrUnscaledIn;
END_GET
SET
lrUnscaledIn:=P_VALUE;
END_SET
END_PROPERTY

PROPERTY P_X_MAX : LREAL
GET
P_X_MAX:=lrX_Max;
END_GET
SET
lrX_Max:=P_X_MAX;
END_SET
END_PROPERTY

PROPERTY P_X_MIN : LREAL
GET
P_X_MIN:=lrX_Min;
END_GET
SET
lrX_Min:=P_X_MIN;
END_SET
END_PROPERTY

PROPERTY P_Y_MAX : LREAL
GET
P_Y_MAX:=lrY_Max;
END_GET
SET
lrY_Max:=P_Y_MAX;
END_SET
END_PROPERTY

PROPERTY P_Y_MIN : LREAL
GET
P_Y_MIN:=lrY_Min;
END_GET
SET
lrY_Min:=P_Y_MIN;
END_SET
END_PROPERTY

END_FUNCTION_BLOCK

// ---- MODULE/BYTES_TO_WORD/VISU/FB_VISU_WORD_TO_BYTES.TcPOU
FUNCTION_BLOCK FB_VISU_WORD_TO_BYTES
VAR_INPUT
END_VAR
VAR_OUTPUT
END_VAR
VAR
	itfOpMode:												I_OP_MODE;
	itfUser:												I_USER_MANAGER;
	itfWordToBytes:											I_WORD_TO_BYTES;
	
	lrUnscaledInput:										LREAL;
	bAdmin:													BOOL;
	bEnable:												BOOL;
END_VAR

VAR PERSISTENT 
	lrXMax:									LREAL:=1;
	lrXMin:                                 LREAL;
	lrYMax:                                 LREAL:=1;
	lrYMin:                                 LREAL;
END_VAR

//Tastensperre bei Auto oder Keiner Betriebsartenauswahl
IF THIS^.itfOpMode.P_OP_MODE_STATE=OP_MODE.MANUAL THEN
	bEnable:=TRUE;
ELSE
	bEnable:=FALSE;
END_IF

bAdmin:=FALSE;
IF itfUser.P_UserGroupID=USER.Admin THEN
	bAdmin:=TRUE;
END_IF
//Übergabe Daten
itfWordToBytes.P_X_MAX:=lrXMax;
itfWordToBytes.P_X_MIN:=lrXMin;
itfWordToBytes.P_Y_MAX:=lrYMax;
itfWordToBytes.P_Y_MIN:=lrYMin;

lrUnscaledInput:=itfWordToBytes.P_VALUE;

METHOD FB_init : BOOL
VAR_INPUT
	bInitRetains : BOOL; // if TRUE, the retain variables are initialized (warm start / cold start)
	bInCopyCode : BOOL;  // if TRUE, the instance afterwards gets moved into the copy code (online change)
	itfOpMode:												I_OP_MODE;
	itfUser:												I_USER_MANAGER;
	itfWordToBytes:											I_WORD_TO_BYTES;
END_VAR
THIS^.itfOpMode:=itfOpMode;
THIS^.itfUser:=itfUser;
THIS^.itfWordToBytes:=itfWordToBytes;
END_METHOD

END_FUNCTION_BLOCK

// ---- MODULE/DATABASE/POU/FB_INFLUX_DB.TcPOU
FUNCTION_BLOCK FB_INFLUX_DB IMPLEMENTS I_DATABASE
VAR //General
	{attribute 'instance-path'} 
  {attribute 'noinit'} 
	strInstancePath:									                      STRING;
	bInit: 												                          BOOL:=TRUE;
	strFullObjectPath: 								                      STRING;
	stEvent:											                          ST_EVENT;
	bAck:												                            BOOL;
	
END_VAR
VAR   // From FB_init	
	itfLogEvents: 										                      I_HANDLE_EVENTS;
  itfOpMode:											                        I_OP_MODE; 
END_VAR                                      				
VAR	// Step chain control                				
  eSeq, eLastSeq, eNextSeq:					                      E_SEQ_DATABASE; 
                  				
  //eActiveSeqState, eLastActiveSeqState:                 E_SEQ_GENERAL;
	(*
  iInternalSeqStateCase, iLastInternalSeqStateCase:       INT:=0;       
	tonDelay, tonTimeOut, tonStepTime:						          TON;
	tDelay:													                        TIME := T#100MS;
	tTimeOut:												                        TIME := T#100MS;
	tTimeOutExt:											                      TIME := T#100MS;
	bDelayActive, bTimeOutActiveQuit, bTimeOutActiveNoQuit:	BOOL;//Timer Option
	bActiveStep, bDebugAcitve, bDebugNext:					        BOOL;//Debug Option
	i:														                          INT;
 	iError:													                        INT; //ERROR-CODE                    	                   		
	listLastSteps:											                    ARRAY[0..49] OF ST_LAST_STEPS;	
	strExtraInfo:											                      STRING; 
	eStep_Type:												                      E_STEP_STATE_TYPE; 
	bDebugModeActive:										                    BOOL;   
	bWaitForBreakpoint:										                  BOOL;
	bBreakpointActive:										                  BOOL;
	bDebugResume:											                      BOOL;   
	listBreakpoint:											                    ARRAY[0..10] OF  INT;    
*)
i:														                            INT;
stSeqCtrlGeneral:											                    ST_SEQ_CTRL_GEN;     	
END_VAR                                             		
VAR                                                 		
	bMethodeFromExtStarted:									                BOOL;
	bMethodeFromExtActive:									                BOOL;
	bMethodeFromExtDone:									                  BOOL;
	strTemp:												                        STRING;
END_VAR   
VAR
  fbSQLDatabase:            FB_SQLDatabaseEvt(sNetID := '', tTimeout := T#5S);
  fbSQLCommand:             FB_SQLCommandEvt(sNetID := '', tTimeout := T#5S);
  fbPLCDBCmd:               FB_PLCDBCmdEvt(sNetID := '', tTimeout := T#5S);
  fbPLCDBCreateEvt:         FB_PLCDBCreateEvt(sNetID := '', tTimeout := T#5S);
  fbPLCDBReadEvt:           FB_PLCDBReadEvt(sNetID:= '', tTimeout:= T#5S);
  fbPLCDBWriteEvt:          FB_PLCDBWriteEvt(sNetID := '', tTimeout := T#5S);
  udiDBID:                  UDINT;
  pDBID:                    POINTER TO UDINT;
  sCmd:                     STRING(5000);
  sTableName:               T_MaxString;
  sDBSymbolName:            STRING;
  pRecord:                  POINTER TO BYTE;
  cbRecord:                 UDINT;
  pValue:                   POINTER TO BYTE;
  cbValue:                  UDINT;
  pColumnNames:             POINTER TO ARRAY [0..MAX_DBCOLUMNS] OF STRING(50);
  cbColumnNames:            UDINT;
  pTableCfg:                POINTER TO ARRAY[0..MAX_DBCOLUMNS] OF ST_ColumnInfo;
  cbTableCfg:               UDINT;
  sOrderByColumn:           STRING(50);
  eOrderBy:                 E_OrderColumn;
  eOrderType:               E_OrderType;
  nStartIndex:              UDINT;
  nRecordCount:             UDINT;
  pData:                    POINTER TO BYTE;
  pData2:                   POINTER TO ST_StandardRecord;
  cbData:                   UDINT;
  pDatabaseConfig:          POINTER TO BYTE;
  cbDatabaseConfig:         UDINT;
  bCreateXMLConfig:         BOOL;
  sColumnNameToUpdate:      STRING;
  sColumnValToUpdate:       STRING;
  sColumnNameToSet:         STRING;
  sNewVal:                  STRING;
  eDBWriteMode:             E_WriteMode;
  nRingBuffParameter:       UDINT;
  stADSDevice:              ST_ADSDevice;
  stSymbol:                 ST_Symbol;
  pExpression:              POINTER TO BYTE;
  cbExpression:             UDINT;
  pParameter:               POINTER TO ARRAY[0..MAX_DBCOLUMNS] OF ST_ExpParameter;
  cbParameter:              UDINT; 
  pSQLCmd:                  POINTER TO BYTE;
  cbSQLCmd:                 UDINT;
  bResult:                  BOOL;
  // Delete table
  fbTaskTableDelete:				NT_StartProcess;
	bDeleteTable:							BOOL;
END_VAR                  	
VAR_TEMP                    	
	iTemp:										INT;
END_VAR

// Set FBs and Interfaces ready after switch internal step
IF stSeqCtrlGeneral.iInternalSeqStateCase <> stSeqCtrlGeneral.iLastInternalSeqStateCase AND NOT stSeqCtrlGeneral.bExitSetReadyState THEN
  IF TRUE
  THEN
    stSeqCtrlGeneral.bExitSetReadyState := TRUE;
  ELSE
    RETURN;
  END_IF
END_IF

stSeqCtrlGeneral.strObject := F_CreateObjectName(strInstancePath);

// First method call
_m_SequenceManager();
//_m_SaveLastStep();

// Actions
A_010_DeleteTable();

CASE eSeq OF 
  E_SEQ_DATABASE.BASE:;
  
	E_SEQ_DATABASE.INIT: _m_Seq_INIT();
		IF TRUE
		AND (stSeqCtrlGeneral.eActiveSeqState = E_SEQ_GENERAL.DONE) 
		THEN
			eSeq := E_SEQ_DATABASE.BASE;
		END_IF
		
	E_SEQ_DATABASE.SETUP:;
  
	// Process
  E_SEQ_DATABASE.CREATE_DATABASE: _m_Seq_CREATE_DATABASE();
    IF TRUE
		AND (stSeqCtrlGeneral.eActiveSeqState = E_SEQ_GENERAL.DONE) 
		THEN
			eSeq := E_SEQ_DATABASE.BASE;
		END_IF
  
	E_SEQ_DATABASE.CONNECT:         _m_Seq_CONNECT();
    IF TRUE
		AND (stSeqCtrlGeneral.eActiveSeqState = E_SEQ_GENERAL.DONE) 
		THEN
			eSeq := E_SEQ_DATABASE.BASE;
		END_IF
    
  E_SEQ_DATABASE.EXECUTE_SIMPLIFY_CMD:  _m_Seq_EXECUTE_SIMPLIFY_CMD();
    IF TRUE
		AND (stSeqCtrlGeneral.eActiveSeqState = E_SEQ_GENERAL.DONE) 
		THEN
			eSeq := E_SEQ_DATABASE.BASE;
		END_IF
  
  E_SEQ_DATABASE.EXECUTE_CMD:     _m_Seq_EXECUTE_CMD();
    IF TRUE
		AND (stSeqCtrlGeneral.eActiveSeqState = E_SEQ_GENERAL.DONE) 
		THEN
			eSeq := E_SEQ_DATABASE.BASE;
		END_IF
    
  E_SEQ_DATABASE.TABLE_EXIST_CHECK:     _m_Seq_TABLE_EXIST_CHECK();
    IF TRUE
		AND (stSeqCtrlGeneral.eActiveSeqState = E_SEQ_GENERAL.DONE) 
		THEN
			eSeq := E_SEQ_DATABASE.BASE;
		END_IF
  
  E_SEQ_DATABASE.CREATE_TABLE:    _m_Seq_CREATE_TABLE();
    IF TRUE
		AND (stSeqCtrlGeneral.eActiveSeqState = E_SEQ_GENERAL.DONE) 
		THEN
			eSeq := E_SEQ_DATABASE.BASE;
		END_IF
  
  E_SEQ_DATABASE.WRITE:           _m_Seq_WRITE();
    IF TRUE
		AND (stSeqCtrlGeneral.eActiveSeqState = E_SEQ_GENERAL.DONE) 
		THEN
			eSeq := E_SEQ_DATABASE.BASE;
		END_IF
  
  E_SEQ_DATABASE.WRITE_STRUCT:    _m_Seq_WRITE_STRUCT();
    IF TRUE
		AND (stSeqCtrlGeneral.eActiveSeqState = E_SEQ_GENERAL.DONE) 
		THEN
			eSeq := E_SEQ_DATABASE.BASE;
		END_IF
  
  E_SEQ_DATABASE.WRITE_BY_SYMBOL: _m_Seq_WRITE_BY_SYMBOL();
    IF TRUE
		AND (stSeqCtrlGeneral.eActiveSeqState = E_SEQ_GENERAL.DONE) 
		THEN
			eSeq := E_SEQ_DATABASE.BASE;
		END_IF
  
  E_SEQ_DATABASE.OVERWRITE:       _m_Seq_OVERWRITE();
    IF TRUE
		AND (stSeqCtrlGeneral.eActiveSeqState = E_SEQ_GENERAL.DONE) 
		THEN
			eSeq := E_SEQ_DATABASE.BASE;
		END_IF
  
  E_SEQ_DATABASE.READ:            _m_Seq_READ();
    IF TRUE
		AND (stSeqCtrlGeneral.eActiveSeqState = E_SEQ_GENERAL.DONE) 
		THEN
			eSeq := E_SEQ_DATABASE.BASE;
		END_IF
  
  E_SEQ_DATABASE.READ_STRUCT:     _m_Seq_READ_STRUCT();
    IF TRUE
		AND (stSeqCtrlGeneral.eActiveSeqState = E_SEQ_GENERAL.DONE) 
		THEN
			eSeq := E_SEQ_DATABASE.BASE;
		END_IF
  
  E_SEQ_DATABASE.CLEAR_TABLE:     _m_Seq_CLEAR_TABLE();
    IF TRUE
		AND (stSeqCtrlGeneral.eActiveSeqState = E_SEQ_GENERAL.DONE) 
		THEN
			eSeq := E_SEQ_DATABASE.BASE;
		END_IF
  
  E_SEQ_DATABASE.DELETE_TABLE:    this^._m_Seq_DELETE_TABLE();
    IF TRUE
		AND (stSeqCtrlGeneral.eActiveSeqState = E_SEQ_GENERAL.DONE) 
		THEN
			eSeq := E_SEQ_DATABASE.BASE;
		END_IF
  
  E_SEQ_DATABASE.DISCONNECT:      _m_Seq_DISCONNECT();
    IF TRUE
		AND (stSeqCtrlGeneral.eActiveSeqState = E_SEQ_GENERAL.DONE) 
		THEN
			eSeq := E_SEQ_DATABASE.BASE;
		END_IF

  // End
	E_SEQ_DATABASE.END:;
	E_SEQ_DATABASE.ERROR_SEQ:;	
END_CASE

strTemp:=TO_STRING(eSeq);

METHOD PRIVATE _m_DebugManager
VAR_INPUT
	iStepID: int;
END_VAR
IF TRUE
AND THIS^.stSeqCtrlGeneral.bDebugModeActive 
AND NOT THIS^.stSeqCtrlGeneral.bActiveStep
THEN


THIS^.stSeqCtrlGeneral.bBreakpointActive:=FALSE;

FOR i:=0 TO 10 DO
	
	IF TRUE
	AND iStepID=THIS^.stSeqCtrlGeneral.listBreakpoint[i] 
	AND iStepID<>0
	THEN
		EXIT;
	END_IF
END_FOR
IF (i<=10) THEN
	THIS^.stSeqCtrlGeneral.bBreakpointActive:=TRUE;
END_IF

END_IF
END_METHOD

METHOD PRIVATE _m_Delay : BOOL
VAR_INPUT
	DelayTime:	TIME;
END_VAR
THIS^.stSeqCtrlGeneral.bDelayActive:=TRUE;
THIS^.stSeqCtrlGeneral.tDelay:=DelayTime;
_m_Delay:=FALSE;
IF THIS^.stSeqCtrlGeneral.tonDelay.Q THEN
	_m_Delay:=TRUE;
END_IF
END_METHOD

METHOD PRIVATE _m_GeneralStepSetting : BOOL
VAR_INPUT
	StepType:			    	E_STEP_STATE_TYPE;
	InfoTextID:					STRING(20);
	EnableDebug:	   			BOOL;	
	
END_VAR
IF THIS^.stSeqCtrlGeneral.bActiveStep THEN
	THIS^.stSeqCtrlGeneral.eStep_Type:=StepType;
	THIS^.stSeqCtrlGeneral.strExtraInfo:= GenLib.F_RET_TXTLIST_ENTRY(strPortNr:='851',strID:='',strTxtLstName:=InfoTextID);
END_IF
END_METHOD

METHOD PRIVATE _m_SaveLastStep : BOOL
VAR_INPUT
END_VAR
VAR
	i: dint;
END_VAR
IF NOT THIS^.stSeqCtrlGeneral.bActiveStep THEN
	
	FOR i:=49 TO 1 BY -1 DO
			stSeqCtrlGeneral.listLastSteps[i].strStepName:=stSeqCtrlGeneral.listLastSteps[i-1].strStepName;
			stSeqCtrlGeneral.listLastSteps[i].tStepTime:=stSeqCtrlGeneral.listLastSteps[i-1].tStepTime;
			stSeqCtrlGeneral.listLastSteps[i].tDelayTime:=stSeqCtrlGeneral.listLastSteps[i-1].tDelayTime;
	END_FOR
	stSeqCtrlGeneral.listLastSteps[0].strStepName:=TO_STRING(THIS^.eSeq);
	stSeqCtrlGeneral.listLastSteps[1].tStepTime:=THIS^.stSeqCtrlGeneral.tonStepTime.ET;
	stSeqCtrlGeneral.listLastSteps[1].tStepTime:=THIS^.stSeqCtrlGeneral.tonDelay.ET;
ELSE
	stSeqCtrlGeneral.listLastSteps[0].tStepTime:=THIS^.stSeqCtrlGeneral.tonStepTime.ET;
	stSeqCtrlGeneral.listLastSteps[0].tDelayTime:=THIS^.stSeqCtrlGeneral.tonDelay.ET;	
END_IF
END_METHOD

METHOD PRIVATE _m_Seq_CLEAR_TABLE : E_SEQ_PROCESS
VAR_INPUT
END_VAR
VAR
	ActiveSeq: STRING;
END_VAR
VAR
	
END_VAR
//THIS^._m_GeneralStepSetting(StepType:=E_STEP_STATE_TYPE.INIT,
ActiveSeq := TO_STRING(THIS^.eSeq);

CASE THIS^.stSeqCtrlGeneral.eActiveSeqState OF
E_SEQ_GENERAL.READY:;

	
E_SEQ_GENERAL.EXECUTE:;
	IF TRUE
	THEN
		THIS^.stSeqCtrlGeneral.eActiveSeqState := E_SEQ_GENERAL.RESET;
	END_IF
  
E_SEQ_GENERAL.RESET:;
	stSeqCtrlGeneral.iInternalSeqStateCase := 0;
	IF TRUE
	THEN
		THIS^.stSeqCtrlGeneral.eActiveSeqState := E_SEQ_GENERAL.BUSY;
	END_IF
  
E_SEQ_GENERAL.BUSY:;
	CASE THIS^.stSeqCtrlGeneral.iInternalSeqStateCase OF
    0:  // Connect to database
      IF TRUE 
      AND NOT THIS^.fbSQLDatabase.bConnected
			THEN 
        IF THIS^.fbSQLDatabase.Connect(THIS^.udiDBID) THEN
          IF THIS^.fbSQLDatabase.bError THEN
            THIS^.stSeqCtrlGeneral.eActiveSeqState := E_SEQ_GENERAL.ERROR;
          ELSE
            THIS^.stSeqCtrlGeneral.iInternalSeqStateCase := 10;
          END_IF
        END_IF
      ELSE
        THIS^.stSeqCtrlGeneral.iInternalSeqStateCase := 10;
			END_IF
      
		10:	// Create command
      IF TRUE 
			THEN 
        sCmd := 'DELETE FROM `';
        sCmd := CONCAT(sCmd, sTableName);
        sCmd := CONCAT(sCmd, '`');
        IF fbSQLDatabase.CreateCmd(ADR(fbSQLCommand)) THEN
          IF fbSqlDatabase.bError THEN
            THIS^.stSeqCtrlGeneral.eActiveSeqState := E_SEQ_GENERAL.ERROR;
          ELSE
            THIS^.stSeqCtrlGeneral.iInternalSeqStateCase := 20;  
          END_IF
        END_IF
			END_IF
      
		20: // Execute command
      IF TRUE 
			THEN
        IF fbSQLCommand.Execute(ADR(sCmd), SIZEOF(sCmd)) THEN
          IF fbSQLCommand.bError THEN
            THIS^.stSeqCtrlGeneral.eActiveSeqState := E_SEQ_GENERAL.ERROR;
          ELSE
            THIS^.stSeqCtrlGeneral.iInternalSeqStateCase := 30;
          END_IF
	      END_IF
			END_IF
      
    30:	// Disconnect
      IF TRUE 
			THEN 
        IF fbSQLDatabase.Disconnect() THEN
          IF fbSqlDatabase.bError THEN
            THIS^.stSeqCtrlGeneral.eActiveSeqState := E_SEQ_GENERAL.ERROR;
          ELSE
            THIS^.stSeqCtrlGeneral.iInternalSeqStateCase := 1000;
          END_IF
        END_IF
			END_IF
      
	ELSE
		THIS^.stSeqCtrlGeneral.eActiveSeqState := E_SEQ_GENERAL.DONE;  
	END_CASE
	THIS^.stSeqCtrlGeneral.strExtraInfo := CONCAT('Internal state: ', TO_STRING(THIS^.stSeqCtrlGeneral.iInternalSeqStateCase));

E_SEQ_GENERAL.DONE:;

E_SEQ_GENERAL.ERROR:;

E_SEQ_GENERAL.TIME_OUT:; 
IF TRUE
AND THIS^.stSeqCtrlGeneral.bTimeOutActiveQuit 
THEN
  THIS^.stSeqCtrlGeneral.strExtraInfo := 'Bitte quittieren und erneut testen';
  IF TRUE
  //AND itfOpMode.P_QUIT
  THEN
    THIS^.stSeqCtrlGeneral.eActiveSeqState := E_SEQ_GENERAL.EXECUTE;
	END_IF
  
END_IF

ELSE
  THIS^.stSeqCtrlGeneral.eActiveSeqState := E_SEQ_GENERAL.ERROR;
END_CASE
END_METHOD

METHOD PRIVATE _m_Seq_CONNECT : E_SEQ_PROCESS
VAR_INPUT
END_VAR
VAR
	ActiveSeq: STRING;
END_VAR
VAR
	
END_VAR
//THIS^._m_GeneralStepSetting(StepType:=E_STEP_STATE_TYPE.INIT,
ActiveSeq := TO_STRING(THIS^.eSeq);

CASE THIS^.stSeqCtrlGeneral.eActiveSeqState OF
E_SEQ_GENERAL.READY:;

	
E_SEQ_GENERAL.EXECUTE:;
	IF TRUE
	THEN
		THIS^.stSeqCtrlGeneral.eActiveSeqState := E_SEQ_GENERAL.RESET;
	END_IF
  
E_SEQ_GENERAL.RESET:;
	stSeqCtrlGeneral.iInternalSeqStateCase := 0;
	IF TRUE
	THEN
		THIS^.stSeqCtrlGeneral.eActiveSeqState := E_SEQ_GENERAL.BUSY;
	END_IF
  
E_SEQ_GENERAL.BUSY:;
	CASE THIS^.stSeqCtrlGeneral.iInternalSeqStateCase OF
		0:	// Entrance step --> Connect
      IF TRUE 
      AND NOT THIS^.fbSQLDatabase.bConnected
			THEN 
        IF THIS^.fbSQLDatabase.Connect(THIS^.udiDBID) THEN
          IF THIS^.fbSQLDatabase.bError THEN
            THIS^.stSeqCtrlGeneral.eActiveSeqState := E_SEQ_GENERAL.ERROR;
          ELSE
            THIS^.stSeqCtrlGeneral.iInternalSeqStateCase := 1000;
          END_IF
        END_IF
      ELSE
        THIS^.stSeqCtrlGeneral.iInternalSeqStateCase := 1000;
			END_IF
      
	ELSE
		THIS^.stSeqCtrlGeneral.eActiveSeqState := E_SEQ_GENERAL.DONE;  
	END_CASE
	THIS^.stSeqCtrlGeneral.strExtraInfo := CONCAT('Internal state: ', TO_STRING(THIS^.stSeqCtrlGeneral.iInternalSeqStateCase));

E_SEQ_GENERAL.DONE:;

E_SEQ_GENERAL.ERROR:;

E_SEQ_GENERAL.TIME_OUT:; 
IF TRUE
AND THIS^.stSeqCtrlGeneral.bTimeOutActiveQuit 
THEN
  THIS^.stSeqCtrlGeneral.strExtraInfo := 'Bitte quittieren und erneut testen';
  IF TRUE
  //AND itfOpMode.P_QUIT
  THEN
    THIS^.stSeqCtrlGeneral.eActiveSeqState := E_SEQ_GENERAL.EXECUTE;
	END_IF
  
END_IF

ELSE
  THIS^.stSeqCtrlGeneral.eActiveSeqState := E_SEQ_GENERAL.ERROR;
END_CASE
END_METHOD

METHOD PRIVATE _m_Seq_CREATE_DATABASE : E_SEQ_PROCESS
VAR_INPUT
END_VAR
VAR
	ActiveSeq: STRING;
END_VAR
VAR
  stTemp:                     STRING;
END_VAR
//THIS^._m_GeneralStepSetting(StepType:=E_STEP_STATE_TYPE.INIT,
ActiveSeq := TO_STRING(THIS^.eSeq);

CASE THIS^.stSeqCtrlGeneral.eActiveSeqState OF
E_SEQ_GENERAL.READY:;

	
E_SEQ_GENERAL.EXECUTE:;
	IF TRUE
	THEN
		THIS^.stSeqCtrlGeneral.eActiveSeqState := E_SEQ_GENERAL.RESET;
	END_IF
  
E_SEQ_GENERAL.RESET:;
	stSeqCtrlGeneral.iInternalSeqStateCase := 0;
	IF TRUE
	THEN
		THIS^.stSeqCtrlGeneral.eActiveSeqState := E_SEQ_GENERAL.BUSY;
	END_IF
  
E_SEQ_GENERAL.BUSY:;
	CASE THIS^.stSeqCtrlGeneral.iInternalSeqStateCase OF
    0:	// Create database
      IF TRUE 
			THEN
        IF fbPLCDBCreateEvt.Database(
          pDatabaseConfig:= pDatabaseConfig,
          cbDatabaseConfig:= cbDatabaseConfig,
          bCreateXMLConfig:= bCreateXMLConfig,
          pDBID := pDBID)
        THEN
          IF fbPLCDBCreateEvt.bError THEN
            THIS^.stSeqCtrlGeneral.eActiveSeqState := E_SEQ_GENERAL.ERROR; 
          ELSE
            THIS^.stSeqCtrlGeneral.iInternalSeqStateCase := 1000;
          END_IF
        END_IF
      END_IF
      
	ELSE
		THIS^.stSeqCtrlGeneral.eActiveSeqState := E_SEQ_GENERAL.DONE;  
	END_CASE
	THIS^.stSeqCtrlGeneral.strExtraInfo := CONCAT('Internal state: ', TO_STRING(THIS^.stSeqCtrlGeneral.iInternalSeqStateCase));

E_SEQ_GENERAL.DONE:;

E_SEQ_GENERAL.ERROR:;

E_SEQ_GENERAL.TIME_OUT:; 
IF TRUE
AND THIS^.stSeqCtrlGeneral.bTimeOutActiveQuit 
THEN
  THIS^.stSeqCtrlGeneral.strExtraInfo := 'Bitte quittieren und erneut testen';
  IF TRUE
  //AND itfOpMode.P_QUIT
  THEN
    THIS^.stSeqCtrlGeneral.eActiveSeqState := E_SEQ_GENERAL.EXECUTE;
	END_IF
  
END_IF

ELSE
  THIS^.stSeqCtrlGeneral.eActiveSeqState := E_SEQ_GENERAL.ERROR;
END_CASE
END_METHOD

METHOD PRIVATE _m_Seq_CREATE_TABLE : E_SEQ_PROCESS
VAR_INPUT
END_VAR
VAR
	ActiveSeq: STRING;
END_VAR
VAR
  stTemp:                     STRING;
END_VAR
//THIS^._m_GeneralStepSetting(StepType:=E_STEP_STATE_TYPE.INIT,
ActiveSeq := TO_STRING(THIS^.eSeq);

CASE THIS^.stSeqCtrlGeneral.eActiveSeqState OF
E_SEQ_GENERAL.READY:;

	
E_SEQ_GENERAL.EXECUTE:;
	IF TRUE
	THEN
		THIS^.stSeqCtrlGeneral.eActiveSeqState := E_SEQ_GENERAL.RESET;
	END_IF
  
E_SEQ_GENERAL.RESET:;
	stSeqCtrlGeneral.iInternalSeqStateCase := 0;
	IF TRUE
	THEN
		THIS^.stSeqCtrlGeneral.eActiveSeqState := E_SEQ_GENERAL.BUSY;
	END_IF
  
E_SEQ_GENERAL.BUSY:;
	CASE THIS^.stSeqCtrlGeneral.iInternalSeqStateCase OF
    0:	// Create table
      IF TRUE 
			THEN
        IF fbPLCDBCreateEvt.Table(hDBID:= udiDBID,
                                  sTableName:= sTableName, 
                                  pTableCfg:= THIS^.pTableCfg, 
                                  cbTableCfg:= THIS^.cbTableCfg)
        THEN
          IF fbPLCDBCreateEvt.bError THEN
            THIS^.stSeqCtrlGeneral.eActiveSeqState := E_SEQ_GENERAL.ERROR; 
          ELSE
            THIS^.stSeqCtrlGeneral.iInternalSeqStateCase := 1000;
          END_IF
        END_IF
      END_IF
      
	ELSE
		THIS^.stSeqCtrlGeneral.eActiveSeqState := E_SEQ_GENERAL.DONE;  
	END_CASE
	THIS^.stSeqCtrlGeneral.strExtraInfo := CONCAT('Internal state: ', TO_STRING(THIS^.stSeqCtrlGeneral.iInternalSeqStateCase));

E_SEQ_GENERAL.DONE:;

E_SEQ_GENERAL.ERROR:;

E_SEQ_GENERAL.TIME_OUT:; 
IF TRUE
AND THIS^.stSeqCtrlGeneral.bTimeOutActiveQuit 
THEN
  THIS^.stSeqCtrlGeneral.strExtraInfo := 'Bitte quittieren und erneut testen';
  IF TRUE
  //AND itfOpMode.P_QUIT
  THEN
    THIS^.stSeqCtrlGeneral.eActiveSeqState := E_SEQ_GENERAL.EXECUTE;
	END_IF
  
END_IF

ELSE
  THIS^.stSeqCtrlGeneral.eActiveSeqState := E_SEQ_GENERAL.ERROR;
END_CASE
END_METHOD

METHOD PRIVATE _m_Seq_DELETE_TABLE : E_SEQ_PROCESS
VAR_INPUT
END_VAR
VAR
	ActiveSeq: STRING;
END_VAR
VAR
	
END_VAR
//THIS^._m_GeneralStepSetting(StepType:=E_STEP_STATE_TYPE.INIT,
ActiveSeq := TO_STRING(THIS^.eSeq);

CASE THIS^.stSeqCtrlGeneral.eActiveSeqState OF
E_SEQ_GENERAL.READY:;

	
E_SEQ_GENERAL.EXECUTE:;
	IF TRUE
	THEN
		THIS^.stSeqCtrlGeneral.eActiveSeqState := E_SEQ_GENERAL.RESET;
	END_IF
  
E_SEQ_GENERAL.RESET:;
	stSeqCtrlGeneral.iInternalSeqStateCase := 0;
	IF TRUE
	THEN
		THIS^.stSeqCtrlGeneral.eActiveSeqState := E_SEQ_GENERAL.BUSY;
	END_IF
  
E_SEQ_GENERAL.BUSY:;
	CASE THIS^.stSeqCtrlGeneral.iInternalSeqStateCase OF
    0:  // Start delete command
      IF TRUE 
			THEN 
        THIS^.bDeleteTable := TRUE;
        THIS^.stSeqCtrlGeneral.iInternalSeqStateCase := 1000;
			END_IF
      
    1000: // Exit seq
      IF TRUE
      THEN
        THIS^.stSeqCtrlGeneral.iInternalSeqStateCase := 9999;
			END_IF
      
	ELSE
		THIS^.stSeqCtrlGeneral.eActiveSeqState := E_SEQ_GENERAL.DONE;  
	END_CASE
	THIS^.stSeqCtrlGeneral.strExtraInfo := CONCAT('Internal state: ', TO_STRING(THIS^.stSeqCtrlGeneral.iInternalSeqStateCase));

E_SEQ_GENERAL.DONE:;

E_SEQ_GENERAL.ERROR:;

E_SEQ_GENERAL.TIME_OUT:; 
IF TRUE
AND THIS^.stSeqCtrlGeneral.bTimeOutActiveQuit 
THEN
  THIS^.stSeqCtrlGeneral.strExtraInfo := 'Bitte quittieren und erneut testen';
  IF TRUE
  //AND itfOpMode.P_QUIT
  THEN
    THIS^.stSeqCtrlGeneral.eActiveSeqState := E_SEQ_GENERAL.EXECUTE;
	END_IF
  
END_IF

ELSE
  THIS^.stSeqCtrlGeneral.eActiveSeqState := E_SEQ_GENERAL.ERROR;
END_CASE
END_METHOD

METHOD PRIVATE _m_Seq_DISCONNECT : E_SEQ_PROCESS
VAR_INPUT
END_VAR
VAR
	ActiveSeq: STRING;
END_VAR
VAR
	
END_VAR
//THIS^._m_GeneralStepSetting(StepType:=E_STEP_STATE_TYPE.INIT,
ActiveSeq := TO_STRING(THIS^.eSeq);

CASE THIS^.stSeqCtrlGeneral.eActiveSeqState OF
E_SEQ_GENERAL.READY:;

	
E_SEQ_GENERAL.EXECUTE:;
	IF TRUE
	THEN
		THIS^.stSeqCtrlGeneral.eActiveSeqState := E_SEQ_GENERAL.RESET;
	END_IF
  
E_SEQ_GENERAL.RESET:;
	stSeqCtrlGeneral.iInternalSeqStateCase := 0;
	IF TRUE
	THEN
		THIS^.stSeqCtrlGeneral.eActiveSeqState := E_SEQ_GENERAL.BUSY;
	END_IF
  
E_SEQ_GENERAL.BUSY:;
	CASE THIS^.stSeqCtrlGeneral.iInternalSeqStateCase OF
		0:	// Entrance step --> Disconnect
      IF TRUE 
			THEN 
        IF fbSQLDatabase.Disconnect() THEN
          IF fbSqlDatabase.bError THEN
            THIS^.stSeqCtrlGeneral.eActiveSeqState := E_SEQ_GENERAL.ERROR;
          ELSE
            THIS^.stSeqCtrlGeneral.iInternalSeqStateCase := 1000;
          END_IF
        END_IF
			END_IF
      
	ELSE
		THIS^.stSeqCtrlGeneral.eActiveSeqState := E_SEQ_GENERAL.DONE;  
	END_CASE
	THIS^.stSeqCtrlGeneral.strExtraInfo := CONCAT('Internal state: ', TO_STRING(THIS^.stSeqCtrlGeneral.iInternalSeqStateCase));

E_SEQ_GENERAL.DONE:;

E_SEQ_GENERAL.ERROR:;

E_SEQ_GENERAL.TIME_OUT:; 
IF TRUE
AND THIS^.stSeqCtrlGeneral.bTimeOutActiveQuit 
THEN
  THIS^.stSeqCtrlGeneral.strExtraInfo := 'Bitte quittieren und erneut testen';
  IF TRUE
  //AND itfOpMode.P_QUIT
  THEN
    THIS^.stSeqCtrlGeneral.eActiveSeqState := E_SEQ_GENERAL.EXECUTE;
	END_IF
  
END_IF

ELSE
  THIS^.stSeqCtrlGeneral.eActiveSeqState := E_SEQ_GENERAL.ERROR;
END_CASE
END_METHOD

METHOD PRIVATE _m_Seq_EXECUTE_CMD : E_SEQ_PROCESS
VAR_INPUT
END_VAR
VAR
	ActiveSeq: STRING;
END_VAR
//THIS^._m_GeneralStepSetting(StepType:=E_STEP_STATE_TYPE.INIT,
ActiveSeq := TO_STRING(THIS^.eSeq);

CASE THIS^.stSeqCtrlGeneral.eActiveSeqState OF
E_SEQ_GENERAL.READY:;

	
E_SEQ_GENERAL.EXECUTE:;
	IF TRUE
	THEN
		THIS^.stSeqCtrlGeneral.eActiveSeqState := E_SEQ_GENERAL.RESET;
	END_IF
  
E_SEQ_GENERAL.RESET:;
	stSeqCtrlGeneral.iInternalSeqStateCase := 0;
	IF TRUE
	THEN
		THIS^.stSeqCtrlGeneral.eActiveSeqState := E_SEQ_GENERAL.BUSY;
	END_IF
  
E_SEQ_GENERAL.BUSY:;
	CASE THIS^.stSeqCtrlGeneral.iInternalSeqStateCase OF
    0:	// Execute command
      IF TRUE 
			THEN 
        IF fbPLCDBCmd.Execute(hDBID:= THIS^.udiDBID, 
                              pExpression:= pExpression, 
                              cbExpression:= cbExpression, 
                              pData:= pData, 
                              cbData:= cbData, 
                              pParameter:= pParameter, 
                              cbParameter:= cbParameter) 
        THEN
          IF fbPLCDBWriteEvt.bError THEN
            THIS^.stSeqCtrlGeneral.eActiveSeqState := E_SEQ_GENERAL.ERROR; 
          ELSE
            THIS^.stSeqCtrlGeneral.iInternalSeqStateCase := 1000;
          END_IF
        END_IF
			END_IF
      
	ELSE
		THIS^.stSeqCtrlGeneral.eActiveSeqState := E_SEQ_GENERAL.DONE;  
	END_CASE
	THIS^.stSeqCtrlGeneral.strExtraInfo := CONCAT('Internal state: ', TO_STRING(THIS^.stSeqCtrlGeneral.iInternalSeqStateCase));

E_SEQ_GENERAL.DONE:;

E_SEQ_GENERAL.ERROR:;

E_SEQ_GENERAL.TIME_OUT:; 
IF TRUE
AND THIS^.stSeqCtrlGeneral.bTimeOutActiveQuit 
THEN
  THIS^.stSeqCtrlGeneral.strExtraInfo := 'Bitte quittieren und erneut testen';
  IF TRUE
  //AND itfOpMode.P_QUIT
  THEN
    THIS^.stSeqCtrlGeneral.eActiveSeqState := E_SEQ_GENERAL.EXECUTE;
	END_IF
  
END_IF

ELSE
  THIS^.stSeqCtrlGeneral.eActiveSeqState := E_SEQ_GENERAL.ERROR;
END_CASE
END_METHOD

METHOD PRIVATE _m_Seq_EXECUTE_SIMPLIFY_CMD : E_SEQ_PROCESS
VAR_INPUT
END_VAR
VAR
	ActiveSeq: STRING;
END_VAR
//THIS^._m_GeneralStepSetting(StepType:=E_STEP_STATE_TYPE.INIT,
ActiveSeq := TO_STRING(THIS^.eSeq);

CASE THIS^.stSeqCtrlGeneral.eActiveSeqState OF
E_SEQ_GENERAL.READY:;

	
E_SEQ_GENERAL.EXECUTE:;
	IF TRUE
	THEN
		THIS^.stSeqCtrlGeneral.eActiveSeqState := E_SEQ_GENERAL.RESET;
	END_IF
  
E_SEQ_GENERAL.RESET:;
	stSeqCtrlGeneral.iInternalSeqStateCase := 0;
	IF TRUE
	THEN
		THIS^.stSeqCtrlGeneral.eActiveSeqState := E_SEQ_GENERAL.BUSY;
	END_IF
  
E_SEQ_GENERAL.BUSY:;
	CASE THIS^.stSeqCtrlGeneral.iInternalSeqStateCase OF
    0:  // Connect to database
      IF TRUE 
      AND NOT THIS^.fbSQLDatabase.bConnected
			THEN 
        IF THIS^.fbSQLDatabase.Connect(THIS^.udiDBID) THEN
          IF THIS^.fbSQLDatabase.bError THEN
            THIS^.stSeqCtrlGeneral.eActiveSeqState := E_SEQ_GENERAL.ERROR;
          ELSE
            THIS^.stSeqCtrlGeneral.iInternalSeqStateCase := 10;
          END_IF
        END_IF
      ELSE
        THIS^.stSeqCtrlGeneral.iInternalSeqStateCase := 10;
			END_IF

    10:	// Execute command
      IF TRUE 
			THEN 
        IF fbSQLCommand.Execute(THIS^.pSQLCmd, THIS^.cbSQLCmd) THEN
          IF fbPLCDBWriteEvt.bError THEN
            THIS^.stSeqCtrlGeneral.eActiveSeqState := E_SEQ_GENERAL.ERROR; 
          ELSE
            THIS^.stSeqCtrlGeneral.iInternalSeqStateCase := 20;
          END_IF
        END_IF
			END_IF
      
    20:	// Disconnect
      IF TRUE 
			THEN 
        IF fbSQLDatabase.Disconnect() THEN
          IF fbSqlDatabase.bError THEN
            THIS^.stSeqCtrlGeneral.eActiveSeqState := E_SEQ_GENERAL.ERROR;
          ELSE
            THIS^.stSeqCtrlGeneral.iInternalSeqStateCase := 1000;
          END_IF
        END_IF
			END_IF
      
	ELSE
		THIS^.stSeqCtrlGeneral.eActiveSeqState := E_SEQ_GENERAL.DONE;  
	END_CASE
	THIS^.stSeqCtrlGeneral.strExtraInfo := CONCAT('Internal state: ', TO_STRING(THIS^.stSeqCtrlGeneral.iInternalSeqStateCase));

E_SEQ_GENERAL.DONE:;

E_SEQ_GENERAL.ERROR:;

E_SEQ_GENERAL.TIME_OUT:; 
IF TRUE
AND THIS^.stSeqCtrlGeneral.bTimeOutActiveQuit 
THEN
  THIS^.stSeqCtrlGeneral.strExtraInfo := 'Bitte quittieren und erneut testen';
  IF TRUE
  //AND itfOpMode.P_QUIT
  THEN
    THIS^.stSeqCtrlGeneral.eActiveSeqState := E_SEQ_GENERAL.EXECUTE;
	END_IF
  
END_IF

ELSE
  THIS^.stSeqCtrlGeneral.eActiveSeqState := E_SEQ_GENERAL.ERROR;
END_CASE
END_METHOD

METHOD PRIVATE _m_Seq_INIT : E_SEQ_PROCESS
VAR_INPUT
END_VAR
VAR
	ActiveSeq: STRING;
END_VAR
VAR
	
END_VAR
//THIS^._m_GeneralStepSetting(StepType:=E_STEP_STATE_TYPE.INIT,
ActiveSeq := TO_STRING(THIS^.eSeq);

CASE THIS^.stSeqCtrlGeneral.eActiveSeqState OF
E_SEQ_GENERAL.READY:;

	
E_SEQ_GENERAL.EXECUTE:;
	IF TRUE
	THEN
		THIS^.stSeqCtrlGeneral.eActiveSeqState := E_SEQ_GENERAL.RESET;
	END_IF
E_SEQ_GENERAL.RESET:;
	stSeqCtrlGeneral.iInternalSeqStateCase := 0;
  
	IF TRUE
	THEN
		THIS^.stSeqCtrlGeneral.eActiveSeqState := E_SEQ_GENERAL.BUSY;
	END_IF
E_SEQ_GENERAL.BUSY:;
	CASE THIS^.stSeqCtrlGeneral.iInternalSeqStateCase OF
		0:	// Entrance step
      IF TRUE
			THEN 
				IF fbSQLDatabase.Disconnect() THEN
          IF fbSqlDatabase.bError THEN
            THIS^.stSeqCtrlGeneral.eActiveSeqState := E_SEQ_GENERAL.ERROR;
          ELSE
            THIS^.stSeqCtrlGeneral.iInternalSeqStateCase := 1000;
          END_IF
        END_IF
			END_IF
      
	ELSE
		THIS^.stSeqCtrlGeneral.eActiveSeqState := E_SEQ_GENERAL.DONE;  
	END_CASE
	THIS^.stSeqCtrlGeneral.strExtraInfo := CONCAT('Internal state: ', TO_STRING(THIS^.stSeqCtrlGeneral.iInternalSeqStateCase));
E_SEQ_GENERAL.DONE:;
E_SEQ_GENERAL.ERROR:;
E_SEQ_GENERAL.TIME_OUT:; 

IF TRUE
AND THIS^.stSeqCtrlGeneral.bTimeOutActiveQuit 
THEN
  THIS^.stSeqCtrlGeneral.strExtraInfo := 'Bitte quittieren und erneut testen';
  IF TRUE
  //AND itfOpMode.P_QUIT
  THEN
    THIS^.stSeqCtrlGeneral.eActiveSeqState := E_SEQ_GENERAL.EXECUTE;
	END_IF
  
END_IF

ELSE
  THIS^.stSeqCtrlGeneral.eActiveSeqState := E_SEQ_GENERAL.ERROR;
END_CASE
END_METHOD

METHOD PRIVATE _m_Seq_OVERWRITE : E_SEQ_PROCESS
VAR_INPUT
END_VAR
VAR
	ActiveSeq: STRING;
END_VAR
VAR
	sTableName:                 STRING;
  sColumnNameToUpdate:        STRING;
  sColumnValToUpdate:         STRING;
  sColumnNameToSet:           STRING;
  sNewVal:                    STRING;
END_VAR
//THIS^._m_GeneralStepSetting(StepType:=E_STEP_STATE_TYPE.INIT,
ActiveSeq := TO_STRING(THIS^.eSeq);

CASE THIS^.stSeqCtrlGeneral.eActiveSeqState OF
E_SEQ_GENERAL.READY:;

	
E_SEQ_GENERAL.EXECUTE:;
	IF TRUE
	THEN
		THIS^.stSeqCtrlGeneral.eActiveSeqState := E_SEQ_GENERAL.RESET;
	END_IF
  
E_SEQ_GENERAL.RESET:;
	stSeqCtrlGeneral.iInternalSeqStateCase := 0;
	IF TRUE
	THEN
		THIS^.stSeqCtrlGeneral.eActiveSeqState := E_SEQ_GENERAL.BUSY;
	END_IF
  
E_SEQ_GENERAL.BUSY:;
	CASE THIS^.stSeqCtrlGeneral.iInternalSeqStateCase OF
		0:  // Connect to database
      IF TRUE 
      AND NOT THIS^.fbSQLDatabase.bConnected
			THEN 
        IF THIS^.fbSQLDatabase.Connect(THIS^.udiDBID) THEN
          IF THIS^.fbSQLDatabase.bError THEN
            THIS^.stSeqCtrlGeneral.eActiveSeqState := E_SEQ_GENERAL.ERROR;
          ELSE
            THIS^.stSeqCtrlGeneral.iInternalSeqStateCase := 10;
          END_IF
        END_IF
      ELSE
        THIS^.stSeqCtrlGeneral.iInternalSeqStateCase := 10;
			END_IF

    10:	// Create command
      IF TRUE 
			THEN 
        sCmd := 'SET SQL_SAFE_UPDATES = 0; UPDATE `';
        sCmd := CONCAT(sCmd, THIS^.sTableName);
        sCmd := CONCAT(sCmd, '` SET ');
        sCmd := CONCAT(sCmd, THIS^.sColumnNameToSet);
        sCmd := CONCAT(sCmd, ' = $'');
        sCmd := CONCAT(sCmd, THIS^.sNewVal);
        sCmd := CONCAT(sCmd, '$' WHERE ');
        sCmd := CONCAT(sCmd, THIS^.sColumnNameToUpdate);
        sCmd := CONCAT(sCmd, ' = $'');
        sCmd := CONCAT(sCmd, THIS^.sColumnValToUpdate);
        sCmd := CONCAT(sCmd, '$';');
        IF fbSQLDatabase.CreateCmd(ADR(fbSQLCommand)) THEN
          IF fbSqlDatabase.bError THEN
            THIS^.stSeqCtrlGeneral.eActiveSeqState := E_SEQ_GENERAL.ERROR;
          ELSE
            THIS^.stSeqCtrlGeneral.iInternalSeqStateCase := 20;  
          END_IF
        END_IF
			END_IF
      
		20: // Execute command
      IF TRUE 
			THEN
        IF fbSQLCommand.Execute(ADR(sCmd), SIZEOF(sCmd)) THEN
          IF fbSQLCommand.bError THEN
            THIS^.stSeqCtrlGeneral.eActiveSeqState := E_SEQ_GENERAL.ERROR;
          ELSE
            THIS^.stSeqCtrlGeneral.iInternalSeqStateCase := 30;
          END_IF
	      END_IF
			END_IF
      
    30:	// Disconnect
      IF TRUE 
			THEN 
        IF fbSQLDatabase.Disconnect() THEN
          IF fbSqlDatabase.bError THEN
            THIS^.stSeqCtrlGeneral.eActiveSeqState := E_SEQ_GENERAL.ERROR;
          ELSE
            THIS^.stSeqCtrlGeneral.iInternalSeqStateCase := 1000;
          END_IF
        END_IF
			END_IF
      
	ELSE
		THIS^.stSeqCtrlGeneral.eActiveSeqState := E_SEQ_GENERAL.DONE;  
	END_CASE
	THIS^.stSeqCtrlGeneral.strExtraInfo := CONCAT('Internal state: ', TO_STRING(THIS^.stSeqCtrlGeneral.iInternalSeqStateCase));

E_SEQ_GENERAL.DONE:;

E_SEQ_GENERAL.ERROR:;

E_SEQ_GENERAL.TIME_OUT:; 
IF TRUE
AND THIS^.stSeqCtrlGeneral.bTimeOutActiveQuit 
THEN
  THIS^.stSeqCtrlGeneral.strExtraInfo := 'Bitte quittieren und erneut testen';
  IF TRUE
  //AND itfOpMode.P_QUIT
  THEN
    THIS^.stSeqCtrlGeneral.eActiveSeqState := E_SEQ_GENERAL.EXECUTE;
	END_IF
  
END_IF

ELSE
  THIS^.stSeqCtrlGeneral.eActiveSeqState := E_SEQ_GENERAL.ERROR;
END_CASE
END_METHOD

METHOD PRIVATE _m_Seq_READ : E_SEQ_PROCESS
VAR_INPUT
END_VAR
VAR
	ActiveSeq: STRING;
END_VAR
VAR
	
END_VAR
//THIS^._m_GeneralStepSetting(StepType:=E_STEP_STATE_TYPE.INIT,
ActiveSeq := TO_STRING(THIS^.eSeq);

CASE THIS^.stSeqCtrlGeneral.eActiveSeqState OF
E_SEQ_GENERAL.READY:;

	
E_SEQ_GENERAL.EXECUTE:;
	IF TRUE
	THEN
		THIS^.stSeqCtrlGeneral.eActiveSeqState := E_SEQ_GENERAL.RESET;
	END_IF
  
E_SEQ_GENERAL.RESET:;
	stSeqCtrlGeneral.iInternalSeqStateCase := 0;
	IF TRUE
	THEN
		THIS^.stSeqCtrlGeneral.eActiveSeqState := E_SEQ_GENERAL.BUSY;
	END_IF
  
E_SEQ_GENERAL.BUSY:;
	CASE THIS^.stSeqCtrlGeneral.iInternalSeqStateCase OF
		0:	// Entrance step --> Read struct
      IF TRUE 
			THEN 
        IF fbPLCDBReadEvt.Read(
          hDBID:= THIS^.udiDBID, 
          sTableName:= THIS^.sTableName, 
          sDBSymbolName:= THIS^.sDBSymbolName, 
          eOrderBy:= THIS^.eOrderBy, 
          eOrderType:= THIS^.eOrderType, 
          nStartIndex:= THIS^.nStartIndex, 
          nRecordCount:= THIS^.nRecordCount, 
          pData:= THIS^.pData2, 
          cbData:= THIS^.cbData)
        THEN
          IF fbPLCDBReadEvt.bError THEN
            THIS^.stSeqCtrlGeneral.eActiveSeqState := E_SEQ_GENERAL.ERROR;
          ELSE
            THIS^.stSeqCtrlGeneral.iInternalSeqStateCase := 1000;
          END_IF
        END_IF
			END_IF
      
	ELSE
		THIS^.stSeqCtrlGeneral.eActiveSeqState := E_SEQ_GENERAL.DONE;  
	END_CASE
	THIS^.stSeqCtrlGeneral.strExtraInfo := CONCAT('Internal state: ', TO_STRING(THIS^.stSeqCtrlGeneral.iInternalSeqStateCase));

E_SEQ_GENERAL.DONE:;

E_SEQ_GENERAL.ERROR:;

E_SEQ_GENERAL.TIME_OUT:; 
IF TRUE
AND THIS^.stSeqCtrlGeneral.bTimeOutActiveQuit 
THEN
  THIS^.stSeqCtrlGeneral.strExtraInfo := 'Bitte quittieren und erneut testen';
  IF TRUE
  //AND itfOpMode.P_QUIT
  THEN
    THIS^.stSeqCtrlGeneral.eActiveSeqState := E_SEQ_GENERAL.EXECUTE;
	END_IF
  
END_IF

ELSE
  THIS^.stSeqCtrlGeneral.eActiveSeqState := E_SEQ_GENERAL.ERROR;
END_CASE
END_METHOD

METHOD PRIVATE _m_Seq_READ_STRUCT : E_SEQ_PROCESS
VAR_INPUT
END_VAR
VAR
	ActiveSeq: STRING;
END_VAR
VAR
	
END_VAR
//THIS^._m_GeneralStepSetting(StepType:=E_STEP_STATE_TYPE.INIT,
ActiveSeq := TO_STRING(THIS^.eSeq);

CASE THIS^.stSeqCtrlGeneral.eActiveSeqState OF
E_SEQ_GENERAL.READY:;

	
E_SEQ_GENERAL.EXECUTE:;
	IF TRUE
	THEN
		THIS^.stSeqCtrlGeneral.eActiveSeqState := E_SEQ_GENERAL.RESET;
	END_IF
  
E_SEQ_GENERAL.RESET:;
	stSeqCtrlGeneral.iInternalSeqStateCase := 0;
	IF TRUE
	THEN
		THIS^.stSeqCtrlGeneral.eActiveSeqState := E_SEQ_GENERAL.BUSY;
	END_IF
  
